LIN {X 0,Y 361.861,Z 153.411,A -85,B 0,C 180,E1 -12922.982,E2 -12922.982} C_VEL
LIN {X 0,Y 361.857,Z 153.413,A -85,B 0,C 180,E1 -12926.632,E2 -12926.632} C_VEL
LIN {X 0,Y 361.847,Z 153.408,A -85,B 0,C 180,E1 -12929.67,E2 -12929.67} C_VEL
LIN {X 0,Y 361.854,Z 153.407,A -85,B 0,C 180,E1 -12933.468,E2 -12933.468} C_VEL
LIN {X 0,Y 361.862,Z 153.407,A -85,B 0,C 180,E1 -12937.144,E2 -12937.144} C_VEL
LIN {X 0,Y 361.842,Z 153.411,A -85,B 0,C 180,E1 -12940.72,E2 -12940.72} C_VEL
LIN {X 0,Y 361.871,Z 153.406,A -85,B 0,C 180,E1 -12943.064,E2 -12943.064} C_VEL
LIN {X 0,Y 361.967,Z 153.396,A -85,B 0,C 180,E1 -12946.527,E2 -12946.527} C_VEL
LIN {X 0,Y 361.997,Z 153.394,A -85,B 0,C 180,E1 -12949.938,E2 -12949.938} C_VEL
LIN {X 0,Y 362.125,Z 153.374,A -85,B 0,C 180,E1 -12953.314,E2 -12953.314} C_VEL
LIN {X 0,Y 362.262,Z 153.362,A -85,B 0,C 180,E1 -12957.777,E2 -12957.777} C_VEL
LIN {X 0,Y 362.178,Z 153.368,A -85,B 0,C 180,E1 -12961.112,E2 -12961.112} C_VEL
LIN {X 0,Y 362.268,Z 153.358,A -85,B 0,C 180,E1 -12962.224,E2 -12962.224} C_VEL
LIN {X 0,Y 362.122,Z 153.374,A -85,B 0,C 180,E1 -12966.688,E2 -12966.688} C_VEL
LIN {X 0,Y 362.003,Z 153.391,A -85,B 0,C 180,E1 -12970.063,E2 -12970.063} C_VEL
LIN {X 0,Y 361.985,Z 153.394,A -85,B 0,C 180,E1 -12973.887,E2 -12973.887} C_VEL
LIN {X 0,Y 361.891,Z 153.403,A -85,B 0,C 180,E1 -12978.103,E2 -12978.103} C_VEL
LIN {X 0,Y 361.858,Z 153.41,A -85,B 0,C 180,E1 -12981.656,E2 -12981.656} C_VEL
LIN {X 0,Y 361.884,Z 153.409,A -85,B 0,C 180,E1 -12985.294,E2 -12985.294} C_VEL
LIN {X 0,Y 361.86,Z 153.413,A -85,B 0,C 180,E1 -12989.074,E2 -12989.074} C_VEL
LIN {X 0,Y 361.851,Z 153.414,A -85,B 0,C 180,E1 -12992.945,E2 -12992.945} C_VEL
LIN {X 0,Y 361.868,Z 153.406,A -85,B 0,C 180,E1 -12995.637,E2 -12995.637} C_VEL
LIN {X 0,Y 361.831,Z 153.415,A -85,B 0,C 180,E1 -12999.018,E2 -12999.018} C_VEL
LIN {X 0,Y 361.836,Z 153.415,A -85,B 0,C 180,E1 -13002.83,E2 -13002.83} C_VEL
LIN {X 0,Y 361.817,Z 153.412,A -85,B 0,C 180,E1 -13005.947,E2 -13005.947} C_VEL
LIN {X 0,Y 361.815,Z 153.413,A -85,B 0,C 180,E1 -13009.249,E2 -13009.249} C_VEL
LIN {X 0,Y 361.868,Z 153.408,A -85,B 0,C 180,E1 -13012.982,E2 -13012.982} C_VEL
LIN {X 0,Y 361.862,Z 153.411,A -85,B 0,C 180,E1 -13016.631,E2 -13016.631} C_VEL
LIN {X 0,Y 361.902,Z 153.409,A -85,B 0,C 180,E1 -13020.668,E2 -13020.668} C_VEL
LIN {X 0,Y 361.894,Z 153.433,A -85,B 0,C 180,E1 -13020.775,E2 -13020.775} C_VEL
LIN {X 0,Y 364.474,Z 166.518,A -85,B 0,C 180,E1 -13023.977,E2 -13023.977} C_VEL
LIN {X 0,Y 365.226,Z 170.606,A -85,B 0,C 180,E1 -13024.954,E2 -13024.954} C_VEL
LIN {X 0,Y 364.174,Z 182.944,A -85,B 0,C 180,E1 -13027.691,E2 -13027.691} C_VEL
LIN {X 0,Y 363.842,Z 187.528,A -85,B 0,C 180,E1 -13028.704,E2 -13028.704} C_VEL
LIN {X 0,Y 368.638,Z 221.989,A -85,B 0,C 180,E1 -13029.653,E2 -13029.653} C_VEL
LIN {X 0,Y 367.445,Z 296.055,A -85,B 0,C 180,E1 -13031.133,E2 -13031.133} C_VEL
LIN {X 0,Y 366.835,Z 309.281,A -85,B 0,C 180,E1 -13031.608,E2 -13031.608} C_VEL
LIN {X 0,Y 366.087,Z 321.461,A -85,B 0,C 180,E1 -13032.256,E2 -13032.256} C_VEL
LIN {X 0,Y 365.205,Z 332.949,A -85,B 0,C 180,E1 -13033.078,E2 -13033.078} C_VEL
LIN {X 0,Y 364.195,Z 344.752,A -85,B 0,C 180,E1 -13034.182,E2 -13034.182} C_VEL
LIN {X 0,Y 363.374,Z 355.364,A -85,B 0,C 180,E1 -13035.437,E2 -13035.437} C_VEL
LIN {X 0,Y 362.449,Z 364.896,A -85,B 0,C 180,E1 -13036.83,E2 -13036.83} C_VEL
LIN {X 0,Y 361.592,Z 374.066,A -85,B 0,C 180,E1 -13038.508,E2 -13038.508} C_VEL
LIN {X 0,Y 361.034,Z 381.452,A -85,B 0,C 180,E1 -13040.193,E2 -13040.193} C_VEL
LIN {X 0,Y 360.707,Z 386.445,A -85,B 0,C 180,E1 -13041.597,E2 -13041.597} C_VEL
LIN {X 0,Y 360.486,Z 391.284,A -85,B 0,C 180,E1 -13043.282,E2 -13043.282} C_VEL
LIN {X 0,Y 360.37,Z 394.981,A -85,B 0,C 180,E1 -13044.965,E2 -13044.965} C_VEL
LIN {X 0,Y 360.314,Z 397.642,A -85,B 0,C 180,E1 -13046.645,E2 -13046.645} C_VEL
LIN {X 0,Y 360.321,Z 398.891,A -85,B 0,C 180,E1 -13047.764,E2 -13047.764} C_VEL
LIN {X 0,Y 360.39,Z 399.729,A -85,B 0,C 180,E1 -13048.882,E2 -13048.882} C_VEL
LIN {X 0,Y 360.426,Z 400.127,A -85,B 0,C 180,E1 -13050,E2 -13050} C_VEL
LIN {X 0,Y 360.36,Z 400.131,A -85,B 0,C 180,E1 -13051.117,E2 -13051.117} C_VEL
LIN {X 0,Y 360.299,Z 398.972,A -85,B 0,C 180,E1 -13053.355,E2 -13053.355} C_VEL
LIN {X 0,Y 360.344,Z 397.756,A -85,B 0,C 180,E1 -13054.474,E2 -13054.474} C_VEL
LIN {X 0,Y 360.379,Z 395.538,A -85,B 0,C 180,E1 -13055.961,E2 -13055.961} C_VEL
LIN {X 0,Y 360.659,Z 391.599,A -85,B 0,C 180,E1 -13057.84,E2 -13057.84} C_VEL
LIN {X 0,Y 361.085,Z 386.927,A -85,B 0,C 180,E1 -13059.523,E2 -13059.523} C_VEL
LIN {X 0,Y 361.83,Z 379.903,A -85,B 0,C 180,E1 -13061.484,E2 -13061.484} C_VEL
LIN {X 0,Y 362.895,Z 372.328,A -85,B 0,C 180,E1 -13063.153,E2 -13063.153} C_VEL
LIN {X 0,Y 364.019,Z 363.164,A -85,B 0,C 180,E1 -13064.774,E2 -13064.774} C_VEL
LIN {X 0,Y 365.223,Z 353.139,A -85,B 0,C 180,E1 -13066.202,E2 -13066.202} C_VEL
LIN {X 0,Y 366.549,Z 342.34,A -85,B 0,C 180,E1 -13067.433,E2 -13067.433} C_VEL
LIN {X 0,Y 367.948,Z 330.06,A -85,B 0,C 180,E1 -13068.515,E2 -13068.515} C_VEL
LIN {X 0,Y 369.043,Z 318.085,A -85,B 0,C 180,E1 -13069.323,E2 -13069.323} C_VEL
LIN {X 0,Y 370.045,Z 304.955,A -85,B 0,C 180,E1 -13069.954,E2 -13069.954} C_VEL
LIN {X 0,Y 370.743,Z 291.887,A -85,B 0,C 180,E1 -13070.349,E2 -13070.349} C_VEL
LIN {X 0,Y 371.93,Z 221.499,A -85,B 0,C 180,E1 -13071.775,E2 -13071.775} C_VEL
LIN {X 0,Y 368.049,Z 198.796,A -85,B 0,C 180,E1 -13072.556,E2 -13072.556} C_VEL
LIN {X 0,Y 365.479,Z 186.6,A -85,B 0,C 180,E1 -13073.056,E2 -13073.056} C_VEL
LIN {X 0,Y 366.598,Z 175.915,A -85,B 0,C 180,E1 -13075.493,E2 -13075.493} C_VEL
LIN {X 0,Y 365.089,Z 167.35,A -85,B 0,C 180,E1 -13077.685,E2 -13077.685} C_VEL
LIN {X 0,Y 362.679,Z 156.746,A -85,B 0,C 180,E1 -13080.558,E2 -13080.558} C_VEL
LIN {X 0,Y 361.891,Z 153.408,A -85,B 0,C 180,E1 -13081.516,E2 -13081.516} C_VEL
LIN {X 0,Y 361.876,Z 153.407,A -85,B 0,C 180,E1 -13085.344,E2 -13085.344} C_VEL
LIN {X 0,Y 361.828,Z 153.418,A -85,B 0,C 180,E1 -13089.018,E2 -13089.018} C_VEL
LIN {X 0,Y 361.833,Z 153.416,A -85,B 0,C 180,E1 -13092.829,E2 -13092.829} C_VEL
LIN {X 0,Y 361.815,Z 153.414,A -85,B 0,C 180,E1 -13095.947,E2 -13095.947} C_VEL
LIN {X 0,Y 361.812,Z 153.414,A -85,B 0,C 180,E1 -13099.249,E2 -13099.249} C_VEL
LIN {X 0,Y 361.862,Z 153.409,A -85,B 0,C 180,E1 -13102.981,E2 -13102.981} C_VEL
LIN {X 0,Y 361.859,Z 153.408,A -85,B 0,C 180,E1 -13106.631,E2 -13106.631} C_VEL
LIN {X 0,Y 361.849,Z 153.404,A -85,B 0,C 180,E1 -13109.669,E2 -13109.669} C_VEL
LIN {X 0,Y 361.855,Z 153.401,A -85,B 0,C 180,E1 -13113.467,E2 -13113.467} C_VEL
LIN {X 0,Y 361.856,Z 153.399,A -85,B 0,C 180,E1 -13117.142,E2 -13117.142} C_VEL
LIN {X 0,Y 361.843,Z 153.408,A -85,B 0,C 180,E1 -13120.719,E2 -13120.719} C_VEL
LIN {X 0,Y 361.879,Z 153.403,A -85,B 0,C 180,E1 -13123.063,E2 -13123.063} C_VEL
LIN {X 0,Y 362.001,Z 153.382,A -85,B 0,C 180,E1 -13126.527,E2 -13126.527} C_VEL
LIN {X 0,Y 361.998,Z 153.393,A -85,B 0,C 180,E1 -13129.936,E2 -13129.936} C_VEL
LIN {X 0,Y 362.125,Z 153.371,A -85,B 0,C 180,E1 -13133.312,E2 -13133.312} C_VEL
LIN {X 0,Y 362.267,Z 153.353,A -85,B 0,C 180,E1 -13137.776,E2 -13137.776} C_VEL
LIN {X 0,Y 362.178,Z 153.362,A -85,B 0,C 180,E1 -13141.111,E2 -13141.111} C_VEL
LIN {X 0,Y 362.279,Z 153.353,A -85,B 0,C 180,E1 -13142.223,E2 -13142.223} C_VEL
LIN {X 0,Y 362.126,Z 153.369,A -85,B 0,C 180,E1 -13146.686,E2 -13146.686} C_VEL
LIN {X 0,Y 362.002,Z 153.383,A -85,B 0,C 180,E1 -13150.062,E2 -13150.062} C_VEL
LIN {X 0,Y 361.999,Z 153.386,A -85,B 0,C 180,E1 -13153.898,E2 -13153.898} C_VEL
LIN {X 0,Y 361.929,Z 153.404,A -85,B 0,C 180,E1 -13156.933,E2 -13156.933} C_VEL
LIN {X 0,Y 361.887,Z 153.408,A -85,B 0,C 180,E1 -13160.46,E2 -13160.46} C_VEL
LIN {X 0,Y 361.893,Z 153.407,A -85,B 0,C 180,E1 -13164.112,E2 -13164.112} C_VEL
LIN {X 0,Y 361.941,Z 153.405,A -85,B 0,C 180,E1 -13166.721,E2 -13166.721} C_VEL
LIN {X 0,Y 361.874,Z 153.408,A -85,B 0,C 180,E1 -13170.327,E2 -13170.327} C_VEL
LIN {X 0,Y 361.853,Z 153.413,A -85,B 0,C 180,E1 -13174.28,E2 -13174.28} C_VEL
LIN {X 0,Y 361.862,Z 153.414,A -85,B 0,C 180,E1 -13177.222,E2 -13177.222} C_VEL
LIN {X 0,Y 361.834,Z 153.421,A -85,B 0,C 180,E1 -13180.755,E2 -13180.755} C_VEL
LIN {X 0,Y 361.877,Z 153.565,A -85,B 0,C 180,E1 -13183.963,E2 -13183.963} C_VEL
LIN {X 0,Y 364.155,Z 163.607,A -85,B 0,C 180,E1 -13186.916,E2 -13186.916} C_VEL
LIN {X 0,Y 369.825,Z 177.061,A -85,B 0,C 180,E1 -13187.659,E2 -13187.659} C_VEL
LIN {X 0,Y 372.692,Z 189.395,A -85,B 0,C 180,E1 -13188.144,E2 -13188.144} C_VEL
LIN {X 0,Y 370.937,Z 271.319,A -85,B 0,C 180,E1 -13189.805,E2 -13189.805} C_VEL
LIN {X 0,Y 370.285,Z 284.163,A -85,B 0,C 180,E1 -13190.276,E2 -13190.276} C_VEL
LIN {X 0,Y 369.554,Z 296.511,A -85,B 0,C 180,E1 -13190.953,E2 -13190.953} C_VEL
LIN {X 0,Y 368.588,Z 307.524,A -85,B 0,C 180,E1 -13191.754,E2 -13191.754} C_VEL
LIN {X 0,Y 367.447,Z 318.475,A -85,B 0,C 180,E1 -13192.78,E2 -13192.78} C_VEL
LIN {X 0,Y 366.247,Z 329.044,A -85,B 0,C 180,E1 -13194.027,E2 -13194.027} C_VEL
LIN {X 0,Y 365.011,Z 338.404,A -85,B 0,C 180,E1 -13195.389,E2 -13195.389} C_VEL
LIN {X 0,Y 363.9,Z 346.954,A -85,B 0,C 180,E1 -13196.935,E2 -13196.935} C_VEL
LIN {X 0,Y 362.763,Z 355.098,A -85,B 0,C 180,E1 -13198.786,E2 -13198.786} C_VEL
LIN {X 0,Y 362.019,Z 360.516,A -85,B 0,C 180,E1 -13200.328,E2 -13200.328} C_VEL
LIN {X 0,Y 361.328,Z 365.639,A -85,B 0,C 180,E1 -13202.172,E2 -13202.172} C_VEL
LIN {X 0,Y 360.95,Z 368.647,A -85,B 0,C 180,E1 -13203.591,E2 -13203.591} C_VEL
LIN {X 0,Y 360.697,Z 370.391,A -85,B 0,C 180,E1 -13204.618,E2 -13204.618} C_VEL
LIN {X 0,Y 360.442,Z 372.569,A -85,B 0,C 180,E1 -13206.406,E2 -13206.406} C_VEL
LIN {X 0,Y 360.236,Z 373.739,A -85,B 0,C 180,E1 -13208.243,E2 -13208.243} C_VEL
LIN {X 0,Y 360.228,Z 373.938,A -85,B 0,C 180,E1 -13209.465,E2 -13209.465} C_VEL
LIN {X 0,Y 360.193,Z 373.659,A -85,B 0,C 180,E1 -13210.628,E2 -13210.628} C_VEL
LIN {X 0,Y 360.293,Z 371.928,A -85,B 0,C 180,E1 -13212.901,E2 -13212.901} C_VEL
LIN {X 0,Y 360.531,Z 369.267,A -85,B 0,C 180,E1 -13214.742,E2 -13214.742} C_VEL
LIN {X 0,Y 360.897,Z 364.776,A -85,B 0,C 180,E1 -13216.823,E2 -13216.823} C_VEL
LIN {X 0,Y 361.319,Z 359.013,A -85,B 0,C 180,E1 -13218.784,E2 -13218.784} C_VEL
LIN {X 0,Y 361.905,Z 352.492,A -85,B 0,C 180,E1 -13220.499,E2 -13220.499} C_VEL
LIN {X 0,Y 362.633,Z 344.333,A -85,B 0,C 180,E1 -13222.203,E2 -13222.203} C_VEL
LIN {X 0,Y 363.424,Z 335.995,A -85,B 0,C 180,E1 -13223.616,E2 -13223.616} C_VEL
LIN {X 0,Y 364.387,Z 325.786,A -85,B 0,C 180,E1 -13225.021,E2 -13225.021} C_VEL
LIN {X 0,Y 365.377,Z 314.188,A -85,B 0,C 180,E1 -13226.278,E2 -13226.278} C_VEL
LIN {X 0,Y 366.165,Z 302.906,A -85,B 0,C 180,E1 -13227.244,E2 -13227.244} C_VEL
LIN {X 0,Y 366.78,Z 291.305,A -85,B 0,C 180,E1 -13228.01,E2 -13228.01} C_VEL
LIN {X 0,Y 367.353,Z 278.024,A -85,B 0,C 180,E1 -13228.63,E2 -13228.63} C_VEL
LIN {X 0,Y 367.735,Z 264.328,A -85,B 0,C 180,E1 -13229.027,E2 -13229.027} C_VEL
LIN {X 0,Y 368.978,Z 187.085,A -85,B 0,C 180,E1 -13230.546,E2 -13230.546} C_VEL
LIN {X 0,Y 365.057,Z 166.996,A -85,B 0,C 180,E1 -13231.152,E2 -13231.152} C_VEL
LIN {X 0,Y 363.773,Z 162.901,A -85,B 0,C 180,E1 -13231.315,E2 -13231.315} C_VEL
LIN {X 0,Y 362.669,Z 156.347,A -85,B 0,C 180,E1 -13233.055,E2 -13233.055} C_VEL
LIN {X 0,Y 361.939,Z 153.406,A -85,B 0,C 180,E1 -13233.897,E2 -13233.897} C_VEL
LIN {X 0,Y 361.945,Z 153.396,A -85,B 0,C 180,E1 -13234.765,E2 -13234.765} C_VEL
LIN {X 0,Y 361.37,Z 153.472,A -85,B 0,C 180,E1 -13235.695,E2 -13235.695} C_VEL
LIN {X 0,Y 358.557,Z 153.819,A -85,B 0,C 180,E1 -13237.209,E2 -13237.209} C_VEL
LIN {X 0,Y 356.11,Z 154.124,A -85,B 0,C 180,E1 -13238.433,E2 -13238.433} C_VEL
LIN {X 0,Y 355.041,Z 154.258,A -85,B 0,C 180,E1 -13239.38,E2 -13239.38} C_VEL
LIN {X 0,Y 354.948,Z 154.267,A -85,B 0,C 180,E1 -13239.701,E2 -13239.701} C_VEL
LIN {X 0,Y 354.893,Z 154.275,A -85,B 0,C 180,E1 -13242.582,E2 -13242.582} C_VEL
LIN {X 0,Y 354.823,Z 154.285,A -85,B 0,C 180,E1 -13246.099,E2 -13246.099} C_VEL
LIN {X 0,Y 354.816,Z 154.284,A -85,B 0,C 180,E1 -13248.477,E2 -13248.477} C_VEL
LIN {X 0,Y 354.795,Z 154.288,A -85,B 0,C 180,E1 -13252.109,E2 -13252.109} C_VEL
LIN {X 0,Y 354.79,Z 154.29,A -85,B 0,C 180,E1 -13255.836,E2 -13255.836} C_VEL
LIN {X 0,Y 354.79,Z 154.29,A -85,B 0,C 180,E1 -13259.685,E2 -13259.685} C_VEL
LIN {X 0,Y 354.783,Z 154.288,A -85,B 0,C 180,E1 -13262.334,E2 -13262.334} C_VEL
LIN {X 0,Y 354.815,Z 154.286,A -85,B 0,C 180,E1 -13265.699,E2 -13265.699} C_VEL
LIN {X 0,Y 354.766,Z 154.293,A -85,B 0,C 180,E1 -13269.413,E2 -13269.413} C_VEL
LIN {X 0,Y 354.779,Z 154.293,A -85,B 0,C 180,E1 -13272.867,E2 -13272.867} C_VEL
LIN {X 0,Y 354.761,Z 154.291,A -85,B 0,C 180,E1 -13276.104,E2 -13276.104} C_VEL
LIN {X 0,Y 354.762,Z 154.294,A -85,B 0,C 180,E1 -13279.176,E2 -13279.176} C_VEL
LIN {X 0,Y 354.798,Z 154.289,A -85,B 0,C 180,E1 -13282.405,E2 -13282.405} C_VEL
LIN {X 0,Y 354.807,Z 154.289,A -85,B 0,C 180,E1 -13284.941,E2 -13284.941} C_VEL
LIN {X 0,Y 354.793,Z 154.291,A -85,B 0,C 180,E1 -13288.406,E2 -13288.406} C_VEL
LIN {X 0,Y 354.789,Z 154.288,A -85,B 0,C 180,E1 -13291.614,E2 -13291.614} C_VEL
LIN {X 0,Y 354.803,Z 154.286,A -85,B 0,C 180,E1 -13295.42,E2 -13295.42} C_VEL
LIN {X 0,Y 354.819,Z 154.284,A -85,B 0,C 180,E1 -13299.113,E2 -13299.113} C_VEL
LIN {X 0,Y 354.839,Z 154.283,A -85,B 0,C 180,E1 -13302.718,E2 -13302.718} C_VEL
LIN {X 0,Y 354.911,Z 154.278,A -85,B 0,C 180,E1 -13306.254,E2 -13306.254} C_VEL
LIN {X 0,Y 354.953,Z 154.27,A -85,B 0,C 180,E1 -13309.736,E2 -13309.736} C_VEL
LIN {X 0,Y 355.092,Z 154.25,A -85,B 0,C 180,E1 -13313.181,E2 -13313.181} C_VEL
LIN {X 0,Y 355.223,Z 154.238,A -85,B 0,C 180,E1 -13317.733,E2 -13317.733} C_VEL
LIN {X 0,Y 355.149,Z 154.243,A -85,B 0,C 180,E1 -13321.135,E2 -13321.135} C_VEL
LIN {X 0,Y 355.23,Z 154.234,A -85,B 0,C 180,E1 -13322.268,E2 -13322.268} C_VEL
LIN {X 0,Y 355.088,Z 154.25,A -85,B 0,C 180,E1 -13326.821,E2 -13326.821} C_VEL
LIN {X 0,Y 354.959,Z 154.267,A -85,B 0,C 180,E1 -13330.265,E2 -13330.265} C_VEL
LIN {X 0,Y 354.928,Z 154.272,A -85,B 0,C 180,E1 -13334.006,E2 -13334.006} C_VEL
LIN {X 0,Y 354.849,Z 154.281,A -85,B 0,C 180,E1 -13338.07,E2 -13338.07} C_VEL
LIN {X 0,Y 354.811,Z 154.285,A -85,B 0,C 180,E1 -13342.108,E2 -13342.108} C_VEL
LIN {X 0,Y 354.853,Z 154.28,A -85,B 0,C 180,E1 -13344.577,E2 -13344.577} C_VEL
LIN {X 0,Y 354.801,Z 154.286,A -85,B 0,C 180,E1 -13348.386,E2 -13348.386} C_VEL
LIN {X 0,Y 354.789,Z 154.288,A -85,B 0,C 180,E1 -13352.334,E2 -13352.334} C_VEL
LIN {X 0,Y 354.823,Z 154.284,A -85,B 0,C 180,E1 -13355.698,E2 -13355.698} C_VEL
LIN {X 0,Y 354.772,Z 154.291,A -85,B 0,C 180,E1 -13359.413,E2 -13359.413} C_VEL
LIN {X 0,Y 354.788,Z 154.293,A -85,B 0,C 180,E1 -13362.866,E2 -13362.866} C_VEL
LIN {X 0,Y 354.767,Z 154.291,A -85,B 0,C 180,E1 -13366.103,E2 -13366.103} C_VEL
LIN {X 0,Y 354.768,Z 154.291,A -85,B 0,C 180,E1 -13369.176,E2 -13369.176} C_VEL
LIN {X 0,Y 354.804,Z 154.291,A -85,B 0,C 180,E1 -13372.404,E2 -13372.404} C_VEL
LIN {X 0,Y 354.815,Z 154.286,A -85,B 0,C 180,E1 -13374.941,E2 -13374.941} C_VEL
LIN {X 0,Y 354.797,Z 154.293,A -85,B 0,C 180,E1 -13378.405,E2 -13378.405} C_VEL
LIN {X 0,Y 354.876,Z 154.373,A -85,B 0,C 180,E1 -13380.53,E2 -13380.53} C_VEL
LIN {X 0,Y 357.397,Z 167.225,A -85,B 0,C 180,E1 -13383.739,E2 -13383.739} C_VEL
LIN {X 0,Y 358.221,Z 172.67,A -85,B 0,C 180,E1 -13385.051,E2 -13385.051} C_VEL
LIN {X 0,Y 356.892,Z 187.314,A -85,B 0,C 180,E1 -13388.356,E2 -13388.356} C_VEL
LIN {X 0,Y 361.844,Z 223.24,A -85,B 0,C 180,E1 -13389.355,E2 -13389.355} C_VEL
LIN {X 0,Y 360.61,Z 295.988,A -85,B 0,C 180,E1 -13390.836,E2 -13390.836} C_VEL
LIN {X 0,Y 359.993,Z 309.152,A -85,B 0,C 180,E1 -13391.319,E2 -13391.319} C_VEL
LIN {X 0,Y 359.213,Z 321.297,A -85,B 0,C 180,E1 -13391.978,E2 -13391.978} C_VEL
LIN {X 0,Y 358.23,Z 333.568,A -85,B 0,C 180,E1 -13392.885,E2 -13392.885} C_VEL
LIN {X 0,Y 357.186,Z 345.199,A -85,B 0,C 180,E1 -13394.01,E2 -13394.01} C_VEL
LIN {X 0,Y 356.369,Z 355.446,A -85,B 0,C 180,E1 -13395.258,E2 -13395.258} C_VEL
LIN {X 0,Y 355.482,Z 364.242,A -85,B 0,C 180,E1 -13396.567,E2 -13396.567} C_VEL
LIN {X 0,Y 354.764,Z 372.124,A -85,B 0,C 180,E1 -13397.994,E2 -13397.994} C_VEL
LIN {X 0,Y 354.106,Z 379.808,A -85,B 0,C 180,E1 -13399.71,E2 -13399.71} C_VEL
LIN {X 0,Y 353.651,Z 385.979,A -85,B 0,C 180,E1 -13401.428,E2 -13401.428} C_VEL
LIN {X 0,Y 353.397,Z 390.862,A -85,B 0,C 180,E1 -13403.147,E2 -13403.147} C_VEL
LIN {X 0,Y 353.273,Z 394.6,A -85,B 0,C 180,E1 -13404.864,E2 -13404.864} C_VEL
LIN {X 0,Y 353.237,Z 397.301,A -85,B 0,C 180,E1 -13406.578,E2 -13406.578} C_VEL
LIN {X 0,Y 353.225,Z 398.568,A -85,B 0,C 180,E1 -13407.719,E2 -13407.719} C_VEL
LIN {X 0,Y 353.292,Z 399.434,A -85,B 0,C 180,E1 -13408.86,E2 -13408.86} C_VEL
LIN {X 0,Y 353.33,Z 399.858,A -85,B 0,C 180,E1 -13410,E2 -13410} C_VEL
LIN {X 0,Y 353.261,Z 399.878,A -85,B 0,C 180,E1 -13411.14,E2 -13411.14} C_VEL
LIN {X 0,Y 353.22,Z 398.762,A -85,B 0,C 180,E1 -13413.422,E2 -13413.422} C_VEL
LIN {X 0,Y 353.257,Z 397.574,A -85,B 0,C 180,E1 -13414.564,E2 -13414.564} C_VEL
LIN {X 0,Y 353.274,Z 395.664,A -85,B 0,C 180,E1 -13415.899,E2 -13415.899} C_VEL
LIN {X 0,Y 353.608,Z 391.49,A -85,B 0,C 180,E1 -13417.997,E2 -13417.997} C_VEL
LIN {X 0,Y 354.05,Z 386.871,A -85,B 0,C 180,E1 -13419.714,E2 -13419.714} C_VEL
LIN {X 0,Y 354.861,Z 379.914,A -85,B 0,C 180,E1 -13421.712,E2 -13421.712} C_VEL
LIN {X 0,Y 355.97,Z 372.413,A -85,B 0,C 180,E1 -13423.414,E2 -13423.414} C_VEL
LIN {X 0,Y 357.098,Z 363.665,A -85,B 0,C 180,E1 -13425.019,E2 -13425.019} C_VEL
LIN {X 0,Y 358.412,Z 353.438,A -85,B 0,C 180,E1 -13426.518,E2 -13426.518} C_VEL
LIN {X 0,Y 359.796,Z 342.763,A -85,B 0,C 180,E1 -13427.771,E2 -13427.771} C_VEL
LIN {X 0,Y 361.062,Z 332.443,A -85,B 0,C 180,E1 -13428.734,E2 -13428.734} C_VEL
LIN {X 0,Y 362.288,Z 320.121,A -85,B 0,C 180,E1 -13429.624,E2 -13429.624} C_VEL
LIN {X 0,Y 363.392,Z 307.201,A -85,B 0,C 180,E1 -13430.298,E2 -13430.298} C_VEL
LIN {X 0,Y 364.193,Z 294.662,A -85,B 0,C 180,E1 -13430.731,E2 -13430.731} C_VEL
LIN {X 0,Y 365.577,Z 222.876,A -85,B 0,C 180,E1 -13432.217,E2 -13432.217} C_VEL
LIN {X 0,Y 361.997,Z 201.712,A -85,B 0,C 180,E1 -13432.961,E2 -13432.961} C_VEL
LIN {X 0,Y 358.807,Z 186.375,A -85,B 0,C 180,E1 -13433.584,E2 -13433.584} C_VEL
LIN {X 0,Y 359.748,Z 177.066,A -85,B 0,C 180,E1 -13435.762,E2 -13435.762} C_VEL
LIN {X 0,Y 358.053,Z 168.195,A -85,B 0,C 180,E1 -13438.104,E2 -13438.104} C_VEL
LIN {X 0,Y 355.749,Z 158.105,A -85,B 0,C 180,E1 -13440.907,E2 -13440.907} C_VEL
LIN {X 0,Y 354.852,Z 154.282,A -85,B 0,C 180,E1 -13442.018,E2 -13442.018} C_VEL
LIN {X 0,Y 354.823,Z 154.289,A -85,B 0,C 180,E1 -13445.699,E2 -13445.699} C_VEL
LIN {X 0,Y 354.77,Z 154.294,A -85,B 0,C 180,E1 -13449.412,E2 -13449.412} C_VEL
LIN {X 0,Y 354.785,Z 154.294,A -85,B 0,C 180,E1 -13452.866,E2 -13452.866} C_VEL
LIN {X 0,Y 354.765,Z 154.293,A -85,B 0,C 180,E1 -13456.103,E2 -13456.103} C_VEL
LIN {X 0,Y 354.765,Z 154.291,A -85,B 0,C 180,E1 -13459.175,E2 -13459.175} C_VEL
LIN {X 0,Y 354.8,Z 154.285,A -85,B 0,C 180,E1 -13462.404,E2 -13462.404} C_VEL
LIN {X 0,Y 354.809,Z 154.284,A -85,B 0,C 180,E1 -13464.94,E2 -13464.94} C_VEL
LIN {X 0,Y 354.795,Z 154.287,A -85,B 0,C 180,E1 -13468.405,E2 -13468.405} C_VEL
LIN {X 0,Y 354.798,Z 154.287,A -85,B 0,C 180,E1 -13471.614,E2 -13471.614} C_VEL
LIN {X 0,Y 354.806,Z 154.286,A -85,B 0,C 180,E1 -13475.419,E2 -13475.419} C_VEL
LIN {X 0,Y 354.817,Z 154.285,A -85,B 0,C 180,E1 -13479.112,E2 -13479.112} C_VEL
LIN {X 0,Y 354.846,Z 154.278,A -85,B 0,C 180,E1 -13482.717,E2 -13482.717} C_VEL
LIN {X 0,Y 354.942,Z 154.263,A -85,B 0,C 180,E1 -13486.254,E2 -13486.254} C_VEL
LIN {X 0,Y 354.955,Z 154.271,A -85,B 0,C 180,E1 -13489.735,E2 -13489.735} C_VEL
LIN {X 0,Y 355.09,Z 154.247,A -85,B 0,C 180,E1 -13493.179,E2 -13493.179} C_VEL
LIN {X 0,Y 355.229,Z 154.229,A -85,B 0,C 180,E1 -13497.732,E2 -13497.732} C_VEL
LIN {X 0,Y 355.149,Z 154.237,A -85,B 0,C 180,E1 -13501.133,E2 -13501.133} C_VEL
LIN {X 0,Y 355.242,Z 154.23,A -85,B 0,C 180,E1 -13502.267,E2 -13502.267} C_VEL
LIN {X 0,Y 355.091,Z 154.246,A -85,B 0,C 180,E1 -13506.819,E2 -13506.819} C_VEL
LIN {X 0,Y 354.958,Z 154.26,A -85,B 0,C 180,E1 -13510.264,E2 -13510.264} C_VEL
LIN {X 0,Y 354.944,Z 154.265,A -85,B 0,C 180,E1 -13514.018,E2 -13514.018} C_VEL
LIN {X 0,Y 354.89,Z 154.272,A -85,B 0,C 180,E1 -13518.091,E2 -13518.091} C_VEL
LIN {X 0,Y 354.819,Z 154.282,A -85,B 0,C 180,E1 -13521.417,E2 -13521.417} C_VEL
LIN {X 0,Y 354.86,Z 154.282,A -85,B 0,C 180,E1 -13524.576,E2 -13524.576} C_VEL
LIN {X 0,Y 354.882,Z 154.28,A -85,B 0,C 180,E1 -13527.095,E2 -13527.095} C_VEL
LIN {X 0,Y 354.853,Z 154.283,A -85,B 0,C 180,E1 -13529.678,E2 -13529.678} C_VEL
LIN {X 0,Y 354.805,Z 154.289,A -85,B 0,C 180,E1 -13533.701,E2 -13533.701} C_VEL
LIN {X 0,Y 354.796,Z 154.293,A -85,B 0,C 180,E1 -13536.459,E2 -13536.459} C_VEL
LIN {X 0,Y 354.822,Z 154.286,A -85,B 0,C 180,E1 -13539.423,E2 -13539.423} C_VEL
LIN {X 0,Y 354.845,Z 154.439,A -85,B 0,C 180,E1 -13543.462,E2 -13543.462} C_VEL
LIN {X 0,Y 357.055,Z 163.923,A -85,B 0,C 180,E1 -13546.329,E2 -13546.329} C_VEL
LIN {X 0,Y 363.741,Z 179.666,A -85,B 0,C 180,E1 -13547.24,E2 -13547.24} C_VEL
LIN {X 0,Y 366.304,Z 190.505,A -85,B 0,C 180,E1 -13547.681,E2 -13547.681} C_VEL
LIN {X 0,Y 364.472,Z 271.592,A -85,B 0,C 180,E1 -13549.353,E2 -13549.353} C_VEL
LIN {X 0,Y 363.85,Z 284.02,A -85,B 0,C 180,E1 -13549.814,E2 -13549.814} C_VEL
LIN {X 0,Y 363.09,Z 296.227,A -85,B 0,C 180,E1 -13550.487,E2 -13550.487} C_VEL
LIN {X 0,Y 362.02,Z 307.908,A -85,B 0,C 180,E1 -13551.344,E2 -13551.344} C_VEL
LIN {X 0,Y 360.706,Z 319.796,A -85,B 0,C 180,E1 -13552.492,E2 -13552.492} C_VEL
LIN {X 0,Y 359.414,Z 330.433,A -85,B 0,C 180,E1 -13553.793,E2 -13553.793} C_VEL
LIN {X 0,Y 358.293,Z 338.41,A -85,B 0,C 180,E1 -13554.988,E2 -13554.988} C_VEL
LIN {X 0,Y 357.111,Z 347.022,A -85,B 0,C 180,E1 -13556.561,E2 -13556.561} C_VEL
LIN {X 0,Y 356.107,Z 353.716,A -85,B 0,C 180,E1 -13558.062,E2 -13558.062} C_VEL
LIN {X 0,Y 355.227,Z 359.657,A -85,B 0,C 180,E1 -13559.701,E2 -13559.701} C_VEL
LIN {X 0,Y 354.454,Z 365.017,A -85,B 0,C 180,E1 -13561.584,E2 -13561.584} C_VEL
LIN {X 0,Y 353.95,Z 368.768,A -85,B 0,C 180,E1 -13563.317,E2 -13563.317} C_VEL
LIN {X 0,Y 353.51,Z 371.835,A -85,B 0,C 180,E1 -13565.324,E2 -13565.324} C_VEL
LIN {X 0,Y 353.332,Z 373.104,A -85,B 0,C 180,E1 -13566.559,E2 -13566.559} C_VEL
LIN {X 0,Y 353.19,Z 373.857,A -85,B 0,C 180,E1 -13567.786,E2 -13567.786} C_VEL
LIN {X 0,Y 353.147,Z 374.205,A -85,B 0,C 180,E1 -13569.282,E2 -13569.282} C_VEL
LIN {X 0,Y 353.101,Z 373.47,A -85,B 0,C 180,E1 -13571.43,E2 -13571.43} C_VEL
LIN {X 0,Y 353.195,Z 372.315,A -85,B 0,C 180,E1 -13572.767,E2 -13572.767} C_VEL
LIN {X 0,Y 353.298,Z 371.008,A -85,B 0,C 180,E1 -13573.83,E2 -13573.83} C_VEL
LIN {X 0,Y 353.621,Z 367.944,A -85,B 0,C 180,E1 -13575.615,E2 -13575.615} C_VEL
LIN {X 0,Y 353.925,Z 363.798,A -85,B 0,C 180,E1 -13577.383,E2 -13577.383} C_VEL
LIN {X 0,Y 354.422,Z 357.408,A -85,B 0,C 180,E1 -13579.431,E2 -13579.431} C_VEL
LIN {X 0,Y 355.026,Z 350.686,A -85,B 0,C 180,E1 -13581.12,E2 -13581.12} C_VEL
LIN {X 0,Y 355.74,Z 343.324,A -85,B 0,C 180,E1 -13582.622,E2 -13582.622} C_VEL
LIN {X 0,Y 356.586,Z 334.719,A -85,B 0,C 180,E1 -13584.061,E2 -13584.061} C_VEL
LIN {X 0,Y 357.636,Z 324.029,A -85,B 0,C 180,E1 -13585.492,E2 -13585.492} C_VEL
LIN {X 0,Y 358.642,Z 312.376,A -85,B 0,C 180,E1 -13586.733,E2 -13586.733} C_VEL
LIN {X 0,Y 359.416,Z 300.812,A -85,B 0,C 180,E1 -13587.688,E2 -13587.688} C_VEL
LIN {X 0,Y 360.133,Z 288.368,A -85,B 0,C 180,E1 -13588.463,E2 -13588.463} C_VEL
LIN {X 0,Y 360.637,Z 275.636,A -85,B 0,C 180,E1 -13589.023,E2 -13589.023} C_VEL
LIN {X 0,Y 360.993,Z 260.577,A -85,B 0,C 180,E1 -13589.408,E2 -13589.408} C_VEL
LIN {X 0,Y 362.223,Z 188.056,A -85,B 0,C 180,E1 -13590.858,E2 -13590.858} C_VEL
LIN {X 0,Y 358.417,Z 168.827,A -85,B 0,C 180,E1 -13591.455,E2 -13591.455} C_VEL
LIN {X 0,Y 356.667,Z 163.075,A -85,B 0,C 180,E1 -13591.695,E2 -13591.695} C_VEL
LIN {X 0,Y 355.473,Z 156.829,A -85,B 0,C 180,E1 -13593.401,E2 -13593.401} C_VEL
LIN {X 0,Y 354.893,Z 154.279,A -85,B 0,C 180,E1 -13594.117,E2 -13594.117} C_VEL
LIN {X 0,Y 355.082,Z 154.251,A -85,B 0,C 180,E1 -13596.821,E2 -13596.821} C_VEL
LIN {X 0,Y 354.948,Z 154.267,A -85,B 0,C 180,E1 -13599.701,E2 -13599.701} C_VEL
LIN {X 0,Y 354.262,Z 154.355,A -85,B 0,C 180,E1 -13600.649,E2 -13600.649} C_VEL
LIN {X 0,Y 351.388,Z 154.713,A -85,B 0,C 180,E1 -13602.189,E2 -13602.189} C_VEL
LIN {X 0,Y 348.954,Z 155.017,A -85,B 0,C 180,E1 -13603.435,E2 -13603.435} C_VEL
LIN {X 0,Y 347.897,Z 155.147,A -85,B 0,C 180,E1 -13604.399,E2 -13604.399} C_VEL
LIN {X 0,Y 347.804,Z 155.158,A -85,B 0,C 180,E1 -13604.726,E2 -13604.726} C_VEL
LIN {X 0,Y 347.783,Z 155.161,A -85,B 0,C 180,E1 -13608.239,E2 -13608.239} C_VEL
LIN {X 0,Y 347.754,Z 155.169,A -85,B 0,C 180,E1 -13611.623,E2 -13611.623} C_VEL
LIN {X 0,Y 347.729,Z 155.17,A -85,B 0,C 180,E1 -13615.115,E2 -13615.115} C_VEL
LIN {X 0,Y 347.721,Z 155.171,A -85,B 0,C 180,E1 -13617.702,E2 -13617.702} C_VEL
LIN {X 0,Y 347.733,Z 155.167,A -85,B 0,C 180,E1 -13620.35,E2 -13620.35} C_VEL
LIN {X 0,Y 347.745,Z 155.165,A -85,B 0,C 180,E1 -13624.044,E2 -13624.044} C_VEL
LIN {X 0,Y 347.752,Z 155.169,A -85,B 0,C 180,E1 -13627.323,E2 -13627.323} C_VEL
LIN {X 0,Y 347.694,Z 155.172,A -85,B 0,C 180,E1 -13630.303,E2 -13630.303} C_VEL
LIN {X 0,Y 347.719,Z 155.17,A -85,B 0,C 180,E1 -13633.409,E2 -13633.409} C_VEL
LIN {X 0,Y 347.721,Z 155.172,A -85,B 0,C 180,E1 -13636.688,E2 -13636.688} C_VEL
LIN {X 0,Y 347.7,Z 155.171,A -85,B 0,C 180,E1 -13640.183,E2 -13640.183} C_VEL
LIN {X 0,Y 347.754,Z 155.169,A -85,B 0,C 180,E1 -13642.679,E2 -13642.679} C_VEL
LIN {X 0,Y 347.748,Z 155.165,A -85,B 0,C 180,E1 -13645.957,E2 -13645.957} C_VEL
LIN {X 0,Y 347.736,Z 155.166,A -85,B 0,C 180,E1 -13649.652,E2 -13649.652} C_VEL
LIN {X 0,Y 347.732,Z 155.167,A -85,B 0,C 180,E1 -13653.6,E2 -13653.6} C_VEL
LIN {X 0,Y 347.749,Z 155.168,A -85,B 0,C 180,E1 -13656.16,E2 -13656.16} C_VEL
LIN {X 0,Y 347.741,Z 155.168,A -85,B 0,C 180,E1 -13659.906,E2 -13659.906} C_VEL
LIN {X 0,Y 347.799,Z 155.164,A -85,B 0,C 180,E1 -13662.356,E2 -13662.356} C_VEL
LIN {X 0,Y 347.854,Z 155.155,A -85,B 0,C 180,E1 -13665.97,E2 -13665.97} C_VEL
LIN {X 0,Y 347.892,Z 155.148,A -85,B 0,C 180,E1 -13669.525,E2 -13669.525} C_VEL
LIN {X 0,Y 348.062,Z 155.126,A -85,B 0,C 180,E1 -13673.042,E2 -13673.042} C_VEL
LIN {X 0,Y 348.185,Z 155.114,A -85,B 0,C 180,E1 -13677.687,E2 -13677.687} C_VEL
LIN {X 0,Y 348.12,Z 155.119,A -85,B 0,C 180,E1 -13681.157,E2 -13681.157} C_VEL
LIN {X 0,Y 348.191,Z 155.111,A -85,B 0,C 180,E1 -13682.314,E2 -13682.314} C_VEL
LIN {X 0,Y 348.056,Z 155.127,A -85,B 0,C 180,E1 -13686.959,E2 -13686.959} C_VEL
LIN {X 0,Y 347.899,Z 155.146,A -85,B 0,C 180,E1 -13690.476,E2 -13690.476} C_VEL
LIN {X 0,Y 347.884,Z 155.148,A -85,B 0,C 180,E1 -13694.137,E2 -13694.137} C_VEL
LIN {X 0,Y 347.799,Z 155.158,A -85,B 0,C 180,E1 -13698.242,E2 -13698.242} C_VEL
LIN {X 0,Y 347.768,Z 155.165,A -85,B 0,C 180,E1 -13701.625,E2 -13701.625} C_VEL
LIN {X 0,Y 347.771,Z 155.167,A -85,B 0,C 180,E1 -13705.112,E2 -13705.112} C_VEL
LIN {X 0,Y 347.748,Z 155.17,A -85,B 0,C 180,E1 -13709.016,E2 -13709.016} C_VEL
LIN {X 0,Y 347.74,Z 155.166,A -85,B 0,C 180,E1 -13711.913,E2 -13711.913} C_VEL
LIN {X 0,Y 347.789,Z 155.16,A -85,B 0,C 180,E1 -13715.876,E2 -13715.876} C_VEL
LIN {X 0,Y 347.735,Z 155.172,A -85,B 0,C 180,E1 -13718.796,E2 -13718.796} C_VEL
LIN {X 0,Y 347.747,Z 155.165,A -85,B 0,C 180,E1 -13721.831,E2 -13721.831} C_VEL
LIN {X 0,Y 347.705,Z 155.173,A -85,B 0,C 180,E1 -13725.028,E2 -13725.028} C_VEL
LIN {X 0,Y 347.743,Z 155.169,A -85,B 0,C 180,E1 -13728.399,E2 -13728.399} C_VEL
LIN {X 0,Y 347.76,Z 155.168,A -85,B 0,C 180,E1 -13732.678,E2 -13732.678} C_VEL
LIN {X 0,Y 347.752,Z 155.166,A -85,B 0,C 180,E1 -13735.956,E2 -13735.956} C_VEL
LIN {X 0,Y 347.798,Z 155.164,A -85,B 0,C 180,E1 -13740.045,E2 -13740.045} C_VEL
LIN {X 0,Y 347.874,Z 155.453,A -85,B 0,C 180,E1 -13740.311,E2 -13740.311} C_VEL
LIN {X 0,Y 350.309,Z 167.904,A -85,B 0,C 180,E1 -13743.488,E2 -13743.488} C_VEL
LIN {X 0,Y 351.231,Z 172.968,A -85,B 0,C 180,E1 -13744.744,E2 -13744.744} C_VEL
LIN {X 0,Y 350.188,Z 184.489,A -85,B 0,C 180,E1 -13747.397,E2 -13747.397} C_VEL
LIN {X 0,Y 349.959,Z 186.998,A -85,B 0,C 180,E1 -13747.972,E2 -13747.972} C_VEL
LIN {X 0,Y 355.012,Z 223.054,A -85,B 0,C 180,E1 -13749.023,E2 -13749.023} C_VEL
LIN {X 0,Y 353.756,Z 295.503,A -85,B 0,C 180,E1 -13750.525,E2 -13750.525} C_VEL
LIN {X 0,Y 353.145,Z 308.757,A -85,B 0,C 180,E1 -13751.018,E2 -13751.018} C_VEL
LIN {X 0,Y 352.336,Z 320.946,A -85,B 0,C 180,E1 -13751.689,E2 -13751.689} C_VEL
LIN {X 0,Y 351.449,Z 332.452,A -85,B 0,C 180,E1 -13752.545,E2 -13752.545} C_VEL
LIN {X 0,Y 350.321,Z 344.256,A -85,B 0,C 180,E1 -13753.688,E2 -13753.688} C_VEL
LIN {X 0,Y 349.45,Z 354.026,A -85,B 0,C 180,E1 -13754.876,E2 -13754.876} C_VEL
LIN {X 0,Y 348.54,Z 363.532,A -85,B 0,C 180,E1 -13756.294,E2 -13756.294} C_VEL
LIN {X 0,Y 347.76,Z 371.506,A -85,B 0,C 180,E1 -13757.748,E2 -13757.748} C_VEL
LIN {X 0,Y 347.054,Z 379.275,A -85,B 0,C 180,E1 -13759.499,E2 -13759.499} C_VEL
LIN {X 0,Y 346.576,Z 385.502,A -85,B 0,C 180,E1 -13761.252,E2 -13761.252} C_VEL
LIN {X 0,Y 346.323,Z 390.436,A -85,B 0,C 180,E1 -13763.006,E2 -13763.006} C_VEL
LIN {X 0,Y 346.196,Z 393.747,A -85,B 0,C 180,E1 -13764.503,E2 -13764.503} C_VEL
LIN {X 0,Y 346.161,Z 396.959,A -85,B 0,C 180,E1 -13766.508,E2 -13766.508} C_VEL
LIN {X 0,Y 346.194,Z 399.132,A -85,B 0,C 180,E1 -13768.837,E2 -13768.837} C_VEL
LIN {X 0,Y 346.235,Z 399.588,A -85,B 0,C 180,E1 -13770,E2 -13770} C_VEL
LIN {X 0,Y 346.162,Z 399.627,A -85,B 0,C 180,E1 -13771.163,E2 -13771.163} C_VEL
LIN {X 0,Y 346.143,Z 398.55,A -85,B 0,C 180,E1 -13773.492,E2 -13773.492} C_VEL
LIN {X 0,Y 346.155,Z 397.401,A -85,B 0,C 180,E1 -13774.658,E2 -13774.658} C_VEL
LIN {X 0,Y 346.199,Z 395.726,A -85,B 0,C 180,E1 -13775.885,E2 -13775.885} C_VEL
LIN {X 0,Y 346.551,Z 391.404,A -85,B 0,C 180,E1 -13778.161,E2 -13778.161} C_VEL
LIN {X 0,Y 347.031,Z 386.835,A -85,B 0,C 180,E1 -13779.912,E2 -13779.912} C_VEL
LIN {X 0,Y 347.904,Z 379.946,A -85,B 0,C 180,E1 -13781.95,E2 -13781.95} C_VEL
LIN {X 0,Y 349.062,Z 372.507,A -85,B 0,C 180,E1 -13783.684,E2 -13783.684} C_VEL
LIN {X 0,Y 350.075,Z 364.951,A -85,B 0,C 180,E1 -13785.128,E2 -13785.128} C_VEL
LIN {X 0,Y 351.34,Z 355.832,A -85,B 0,C 180,E1 -13786.562,E2 -13786.562} C_VEL
LIN {X 0,Y 352.808,Z 345.742,A -85,B 0,C 180,E1 -13787.835,E2 -13787.835} C_VEL
LIN {X 0,Y 354.213,Z 334.581,A -85,B 0,C 180,E1 -13788.959,E2 -13788.959} C_VEL
LIN {X 0,Y 355.405,Z 324.056,A -85,B 0,C 180,E1 -13789.794,E2 -13789.794} C_VEL
LIN {X 0,Y 356.551,Z 311.447,A -85,B 0,C 180,E1 -13790.555,E2 -13790.555} C_VEL
LIN {X 0,Y 357.447,Z 299.04,A -85,B 0,C 180,E1 -13791.066,E2 -13791.066} C_VEL
LIN {X 0,Y 357.987,Z 283.584,A -85,B 0,C 180,E1 -13791.447,E2 -13791.447} C_VEL
LIN {X 0,Y 359.134,Z 223.619,A -85,B 0,C 180,E1 -13792.697,E2 -13792.697} C_VEL
LIN {X 0,Y 355.564,Z 202.272,A -85,B 0,C 180,E1 -13793.47,E2 -13793.47} C_VEL
LIN {X 0,Y 352.148,Z 186.078,A -85,B 0,C 180,E1 -13794.161,E2 -13794.161} C_VEL
LIN {X 0,Y 352.866,Z 178.473,A -85,B 0,C 180,E1 -13795.987,E2 -13795.987} C_VEL
LIN {X 0,Y 351.223,Z 169.896,A -85,B 0,C 180,E1 -13798.303,E2 -13798.303} C_VEL
LIN {X 0,Y 348.87,Z 159.542,A -85,B 0,C 180,E1 -13801.247,E2 -13801.247} C_VEL
LIN {X 0,Y 347.773,Z 155.165,A -85,B 0,C 180,E1 -13802.606,E2 -13802.606} C_VEL
LIN {X 0,Y 347.771,Z 155.165,A -85,B 0,C 180,E1 -13806.064,E2 -13806.064} C_VEL
LIN {X 0,Y 347.733,Z 155.172,A -85,B 0,C 180,E1 -13808.795,E2 -13808.795} C_VEL
LIN {X 0,Y 347.744,Z 155.164,A -85,B 0,C 180,E1 -13811.831,E2 -13811.831} C_VEL
LIN {X 0,Y 347.703,Z 155.175,A -85,B 0,C 180,E1 -13815.027,E2 -13815.027} C_VEL
LIN {X 0,Y 347.74,Z 155.17,A -85,B 0,C 180,E1 -13818.399,E2 -13818.399} C_VEL
LIN {X 0,Y 347.763,Z 155.161,A -85,B 0,C 180,E1 -13822.014,E2 -13822.014} C_VEL
LIN {X 0,Y 347.745,Z 155.161,A -85,B 0,C 180,E1 -13825.535,E2 -13825.535} C_VEL
LIN {X 0,Y 347.746,Z 155.166,A -85,B 0,C 180,E1 -13828.3,E2 -13828.3} C_VEL
LIN {X 0,Y 347.746,Z 155.167,A -85,B 0,C 180,E1 -13830.984,E2 -13830.984} C_VEL
LIN {X 0,Y 347.735,Z 155.16,A -85,B 0,C 180,E1 -13833.599,E2 -13833.599} C_VEL
LIN {X 0,Y 347.748,Z 155.166,A -85,B 0,C 180,E1 -13836.158,E2 -13836.158} C_VEL
LIN {X 0,Y 347.765,Z 155.166,A -85,B 0,C 180,E1 -13839.906,E2 -13839.906} C_VEL
LIN {X 0,Y 347.792,Z 155.158,A -85,B 0,C 180,E1 -13843.566,E2 -13843.566} C_VEL
LIN {X 0,Y 347.887,Z 155.138,A -85,B 0,C 180,E1 -13847.16,E2 -13847.16} C_VEL
LIN {X 0,Y 347.936,Z 155.138,A -85,B 0,C 180,E1 -13850.7,E2 -13850.7} C_VEL
LIN {X 0,Y 348.042,Z 155.13,A -85,B 0,C 180,E1 -13854.205,E2 -13854.205} C_VEL
LIN {X 0,Y 348.19,Z 155.104,A -85,B 0,C 180,E1 -13857.686,E2 -13857.686} C_VEL
LIN {X 0,Y 348.121,Z 155.112,A -85,B 0,C 180,E1 -13861.156,E2 -13861.156} C_VEL
LIN {X 0,Y 348.204,Z 155.106,A -85,B 0,C 180,E1 -13862.313,E2 -13862.313} C_VEL
LIN {X 0,Y 348.058,Z 155.122,A -85,B 0,C 180,E1 -13866.958,E2 -13866.958} C_VEL
LIN {X 0,Y 347.898,Z 155.139,A -85,B 0,C 180,E1 -13870.475,E2 -13870.475} C_VEL
LIN {X 0,Y 347.899,Z 155.142,A -85,B 0,C 180,E1 -13874.149,E2 -13874.149} C_VEL
LIN {X 0,Y 347.83,Z 155.151,A -85,B 0,C 180,E1 -13878.259,E2 -13878.259} C_VEL
LIN {X 0,Y 347.768,Z 155.159,A -85,B 0,C 180,E1 -13881.626,E2 -13881.626} C_VEL
LIN {X 0,Y 347.811,Z 155.158,A -85,B 0,C 180,E1 -13885.108,E2 -13885.108} C_VEL
LIN {X 0,Y 347.809,Z 155.158,A -85,B 0,C 180,E1 -13887.693,E2 -13887.693} C_VEL
LIN {X 0,Y 347.763,Z 155.166,A -85,B 0,C 180,E1 -13890.346,E2 -13890.346} C_VEL
LIN {X 0,Y 347.743,Z 155.169,A -85,B 0,C 180,E1 -13894.463,E2 -13894.463} C_VEL
LIN {X 0,Y 347.772,Z 155.169,A -85,B 0,C 180,E1 -13897.988,E2 -13897.988} C_VEL
LIN {X 0,Y 347.749,Z 155.17,A -85,B 0,C 180,E1 -13901.83,E2 -13901.83} C_VEL
LIN {X 0,Y 347.766,Z 155.217,A -85,B 0,C 180,E1 -13902.904,E2 -13902.904} C_VEL
LIN {X 0,Y 349.949,Z 164.359,A -85,B 0,C 180,E1 -13905.708,E2 -13905.708} C_VEL
LIN {X 0,Y 357.65,Z 182.011,A -85,B 0,C 180,E1 -13906.794,E2 -13906.794} C_VEL
LIN {X 0,Y 359.938,Z 191.782,A -85,B 0,C 180,E1 -13907.206,E2 -13907.206} C_VEL
LIN {X 0,Y 358.024,Z 271.814,A -85,B 0,C 180,E1 -13908.883,E2 -13908.883} C_VEL
LIN {X 0,Y 357.331,Z 285.099,A -85,B 0,C 180,E1 -13909.391,E2 -13909.391} C_VEL
LIN {X 0,Y 356.496,Z 297.506,A -85,B 0,C 180,E1 -13910.1,E2 -13910.1} C_VEL
LIN {X 0,Y 355.449,Z 308.441,A -85,B 0,C 180,E1 -13910.932,E2 -13910.932} C_VEL
LIN {X 0,Y 354.117,Z 319.679,A -85,B 0,C 180,E1 -13912.03,E2 -13912.03} C_VEL
LIN {X 0,Y 352.813,Z 329.996,A -85,B 0,C 180,E1 -13913.302,E2 -13913.302} C_VEL
LIN {X 0,Y 351.432,Z 339.506,A -85,B 0,C 180,E1 -13914.75,E2 -13914.75} C_VEL
LIN {X 0,Y 350.339,Z 347.086,A -85,B 0,C 180,E1 -13916.173,E2 -13916.173} C_VEL
LIN {X 0,Y 349.051,Z 355.13,A -85,B 0,C 180,E1 -13918.046,E2 -13918.046} C_VEL
LIN {X 0,Y 348.173,Z 360.774,A -85,B 0,C 180,E1 -13919.693,E2 -13919.693} C_VEL
LIN {X 0,Y 347.377,Z 365.949,A -85,B 0,C 180,E1 -13921.612,E2 -13921.612} C_VEL
LIN {X 0,Y 346.81,Z 369.792,A -85,B 0,C 180,E1 -13923.524,E2 -13923.524} C_VEL
LIN {X 0,Y 346.524,Z 371.664,A -85,B 0,C 180,E1 -13924.792,E2 -13924.792} C_VEL
LIN {X 0,Y 346.319,Z 373.04,A -85,B 0,C 180,E1 -13926.054,E2 -13926.054} C_VEL
LIN {X 0,Y 346.137,Z 373.97,A -85,B 0,C 180,E1 -13927.308,E2 -13927.308} C_VEL
LIN {X 0,Y 346.05,Z 374.46,A -85,B 0,C 180,E1 -13929.101,E2 -13929.101} C_VEL
LIN {X 0,Y 346.019,Z 373.956,A -85,B 0,C 180,E1 -13931.036,E2 -13931.036} C_VEL
LIN {X 0,Y 346.082,Z 372.685,A -85,B 0,C 180,E1 -13932.637,E2 -13932.637} C_VEL
LIN {X 0,Y 346.352,Z 369.933,A -85,B 0,C 180,E1 -13934.705,E2 -13934.705} C_VEL
LIN {X 0,Y 346.684,Z 366.015,A -85,B 0,C 180,E1 -13936.667,E2 -13936.667} C_VEL
LIN {X 0,Y 347.041,Z 361.659,A -85,B 0,C 180,E1 -13938.316,E2 -13938.316} C_VEL
LIN {X 0,Y 347.604,Z 355.651,A -85,B 0,C 180,E1 -13940.104,E2 -13940.104} C_VEL
LIN {X 0,Y 348.335,Z 348.15,A -85,B 0,C 180,E1 -13941.881,E2 -13941.881} C_VEL
LIN {X 0,Y 349.089,Z 340.506,A -85,B 0,C 180,E1 -13943.353,E2 -13943.353} C_VEL
LIN {X 0,Y 350.051,Z 331.22,A -85,B 0,C 180,E1 -13944.817,E2 -13944.817} C_VEL
LIN {X 0,Y 351.035,Z 320.881,A -85,B 0,C 180,E1 -13946.126,E2 -13946.126} C_VEL
LIN {X 0,Y 352.038,Z 308.796,A -85,B 0,C 180,E1 -13947.337,E2 -13947.337} C_VEL
LIN {X 0,Y 352.75,Z 297.532,A -85,B 0,C 180,E1 -13948.216,E2 -13948.216} C_VEL
LIN {X 0,Y 353.399,Z 285.151,A -85,B 0,C 180,E1 -13948.932,E2 -13948.932} C_VEL
LIN {X 0,Y 353.962,Z 272.408,A -85,B 0,C 180,E1 -13949.431,E2 -13949.431} C_VEL
LIN {X 0,Y 354.42,Z 246.752,A -85,B 0,C 180,E1 -13950,E2 -13950} C_VEL
LIN {X 0,Y 355.386,Z 188.745,A -85,B 0,C 180,E1 -13951.187,E2 -13951.187} C_VEL
LIN {X 0,Y 352.033,Z 171.371,A -85,B 0,C 180,E1 -13951.736,E2 -13951.736} C_VEL
LIN {X 0,Y 349.579,Z 163.332,A -85,B 0,C 180,E1 -13952.067,E2 -13952.067} C_VEL
LIN {X 0,Y 347.857,Z 155.153,A -85,B 0,C 180,E1 -13954.418,E2 -13954.418} C_VEL
LIN {X 0,Y 348.05,Z 155.127,A -85,B 0,C 180,E1 -13956.959,E2 -13956.959} C_VEL
LIN {X 0,Y 347.884,Z 155.148,A -85,B 0,C 180,E1 -13960.476,E2 -13960.476} C_VEL
LIN {X 0,Y 347.848,Z 155.155,A -85,B 0,C 180,E1 -13964.119,E2 -13964.119} C_VEL
LIN {X 0,Y 347.804,Z 155.158,A -85,B 0,C 180,E1 -13964.726,E2 -13964.726} C_VEL
LIN {X 0,Y 347.109,Z 155.251,A -85,B 0,C 180,E1 -13965.693,E2 -13965.693} C_VEL
LIN {X 0,Y 344.22,Z 155.607,A -85,B 0,C 180,E1 -13967.266,E2 -13967.266} C_VEL
LIN {X 0,Y 341.788,Z 155.909,A -85,B 0,C 180,E1 -13968.539,E2 -13968.539} C_VEL
LIN {X 0,Y 340.747,Z 156.042,A -85,B 0,C 180,E1 -13969.525,E2 -13969.525} C_VEL
LIN {X 0,Y 340.664,Z 156.046,A -85,B 0,C 180,E1 -13969.859,E2 -13969.859} C_VEL
LIN {X 0,Y 340.693,Z 156.046,A -85,B 0,C 180,E1 -13973.076,E2 -13973.076} C_VEL
LIN {X 0,Y 340.705,Z 156.044,A -85,B 0,C 180,E1 -13976.989,E2 -13976.989} C_VEL
LIN {X 0,Y 340.689,Z 156.047,A -85,B 0,C 180,E1 -13981.046,E2 -13981.046} C_VEL
LIN {X 0,Y 340.712,Z 156.046,A -85,B 0,C 180,E1 -13985.28,E2 -13985.28} C_VEL
LIN {X 0,Y 340.69,Z 156.044,A -85,B 0,C 180,E1 -13988.383,E2 -13988.383} C_VEL
LIN {X 0,Y 340.688,Z 156.044,A -85,B 0,C 180,E1 -13992.045,E2 -13992.045} C_VEL
LIN {X 0,Y 340.648,Z 156.05,A -85,B 0,C 180,E1 -13996.228,E2 -13996.228} C_VEL
LIN {X 0,Y 340.667,Z 156.051,A -85,B 0,C 180,E1 -13998.689,E2 -13998.689} C_VEL
LIN {X 0,Y 340.718,Z 156.04,A -85,B 0,C 180,E1 -14001.772,E2 -14001.772} C_VEL
LIN {X 0,Y 340.722,Z 156.04,A -85,B 0,C 180,E1 -14005.597,E2 -14005.597} C_VEL
LIN {X 0,Y 340.692,Z 156.046,A -85,B 0,C 180,E1 -14008.956,E2 -14008.956} C_VEL
LIN {X 0,Y 340.71,Z 156.043,A -85,B 0,C 180,E1 -14013.013,E2 -14013.013} C_VEL
LIN {X 0,Y 340.701,Z 156.044,A -85,B 0,C 180,E1 -14016.926,E2 -14016.926} C_VEL
LIN {X 0,Y 340.691,Z 156.046,A -85,B 0,C 180,E1 -14020.728,E2 -14020.728} C_VEL
LIN {X 0,Y 340.728,Z 156.039,A -85,B 0,C 180,E1 -14023.216,E2 -14023.216} C_VEL
LIN {X 0,Y 340.817,Z 156.029,A -85,B 0,C 180,E1 -14026.89,E2 -14026.89} C_VEL
LIN {X 0,Y 340.883,Z 156.022,A -85,B 0,C 180,E1 -14030.507,E2 -14030.507} C_VEL
LIN {X 0,Y 341.012,Z 156.004,A -85,B 0,C 180,E1 -14032.898,E2 -14032.898} C_VEL
LIN {X 0,Y 340.811,Z 156.029,A -85,B 0,C 180,E1 -14035.269,E2 -14035.269} C_VEL
LIN {X 0,Y 341.121,Z 155.994,A -85,B 0,C 180,E1 -14037.639,E2 -14037.639} C_VEL
LIN {X 0,Y 341.092,Z 155.995,A -85,B 0,C 180,E1 -14041.181,E2 -14041.181} C_VEL
LIN {X 0,Y 341.128,Z 155.99,A -85,B 0,C 180,E1 -14042.362,E2 -14042.362} C_VEL
LIN {X 0,Y 341.004,Z 156.006,A -85,B 0,C 180,E1 -14047.104,E2 -14047.104} C_VEL
LIN {X 0,Y 340.851,Z 156.024,A -85,B 0,C 180,E1 -14050.695,E2 -14050.695} C_VEL
LIN {X 0,Y 340.823,Z 156.027,A -85,B 0,C 180,E1 -14054.327,E2 -14054.327} C_VEL
LIN {X 0,Y 340.761,Z 156.035,A -85,B 0,C 180,E1 -14058.426,E2 -14058.426} C_VEL
LIN {X 0,Y 340.723,Z 156.041,A -85,B 0,C 180,E1 -14061.842,E2 -14061.842} C_VEL
LIN {X 0,Y 340.719,Z 156.042,A -85,B 0,C 180,E1 -14065.669,E2 -14065.669} C_VEL
LIN {X 0,Y 340.707,Z 156.043,A -85,B 0,C 180,E1 -14069.675,E2 -14069.675} C_VEL
LIN {X 0,Y 340.689,Z 156.045,A -85,B 0,C 180,E1 -14072.436,E2 -14072.436} C_VEL
LIN {X 0,Y 340.72,Z 156.043,A -85,B 0,C 180,E1 -14075.279,E2 -14075.279} C_VEL
LIN {X 0,Y 340.698,Z 156.045,A -85,B 0,C 180,E1 -14078.383,E2 -14078.383} C_VEL
LIN {X 0,Y 340.697,Z 156.043,A -85,B 0,C 180,E1 -14082.044,E2 -14082.044} C_VEL
LIN {X 0,Y 340.654,Z 156.05,A -85,B 0,C 180,E1 -14086.227,E2 -14086.227} C_VEL
LIN {X 0,Y 340.674,Z 156.051,A -85,B 0,C 180,E1 -14088.688,E2 -14088.688} C_VEL
LIN {X 0,Y 340.723,Z 156.04,A -85,B 0,C 180,E1 -14091.771,E2 -14091.771} C_VEL
LIN {X 0,Y 340.727,Z 156.04,A -85,B 0,C 180,E1 -14095.595,E2 -14095.595} C_VEL
LIN {X 0,Y 340.755,Z 156.041,A -85,B 0,C 180,E1 -14099.923,E2 -14099.923} C_VEL
LIN {X 0,Y 343.242,Z 168.576,A -85,B 0,C 180,E1 -14103.227,E2 -14103.227} C_VEL
LIN {X 0,Y 344.255,Z 175.376,A -85,B 0,C 180,E1 -14104.937,E2 -14104.937} C_VEL
LIN {X 0,Y 343.05,Z 186.795,A -85,B 0,C 180,E1 -14107.608,E2 -14107.608} C_VEL
LIN {X 0,Y 348.225,Z 223.682,A -85,B 0,C 180,E1 -14108.698,E2 -14108.698} C_VEL
LIN {X 0,Y 346.937,Z 295.018,A -85,B 0,C 180,E1 -14110.203,E2 -14110.203} C_VEL
LIN {X 0,Y 346.307,Z 308.349,A -85,B 0,C 180,E1 -14110.706,E2 -14110.706} C_VEL
LIN {X 0,Y 345.382,Z 321.703,A -85,B 0,C 180,E1 -14111.461,E2 -14111.461} C_VEL
LIN {X 0,Y 344.476,Z 332.926,A -85,B 0,C 180,E1 -14112.333,E2 -14112.333} C_VEL
LIN {X 0,Y 343.333,Z 344.586,A -85,B 0,C 180,E1 -14113.499,E2 -14113.499} C_VEL
LIN {X 0,Y 342.418,Z 354.348,A -85,B 0,C 180,E1 -14114.724,E2 -14114.724} C_VEL
LIN {X 0,Y 341.616,Z 362.782,A -85,B 0,C 180,E1 -14116.011,E2 -14116.011} C_VEL
LIN {X 0,Y 340.786,Z 370.838,A -85,B 0,C 180,E1 -14117.494,E2 -14117.494} C_VEL
LIN {X 0,Y 340.012,Z 378.706,A -85,B 0,C 180,E1 -14119.279,E2 -14119.279} C_VEL
LIN {X 0,Y 339.522,Z 384.994,A -85,B 0,C 180,E1 -14121.069,E2 -14121.069} C_VEL
LIN {X 0,Y 339.25,Z 389.981,A -85,B 0,C 180,E1 -14122.86,E2 -14122.86} C_VEL
LIN {X 0,Y 339.098,Z 393.671,A -85,B 0,C 180,E1 -14124.57,E2 -14124.57} C_VEL
LIN {X 0,Y 339.086,Z 396.601,A -85,B 0,C 180,E1 -14126.435,E2 -14126.435} C_VEL
LIN {X 0,Y 339.096,Z 398.818,A -85,B 0,C 180,E1 -14128.812,E2 -14128.812} C_VEL
LIN {X 0,Y 339.14,Z 399.316,A -85,B 0,C 180,E1 -14130,E2 -14130} C_VEL
LIN {X 0,Y 339.063,Z 399.376,A -85,B 0,C 180,E1 -14131.187,E2 -14131.187} C_VEL
LIN {X 0,Y 339.066,Z 398.342,A -85,B 0,C 180,E1 -14133.565,E2 -14133.565} C_VEL
LIN {X 0,Y 339.059,Z 397.232,A -85,B 0,C 180,E1 -14134.756,E2 -14134.756} C_VEL
LIN {X 0,Y 339.132,Z 395.675,A -85,B 0,C 180,E1 -14135.947,E2 -14135.947} C_VEL
LIN {X 0,Y 339.356,Z 392.566,A -85,B 0,C 180,E1 -14137.736,E2 -14137.736} C_VEL
LIN {X 0,Y 339.818,Z 388.415,A -85,B 0,C 180,E1 -14139.523,E2 -14139.523} C_VEL
LIN {X 0,Y 340.592,Z 382.099,A -85,B 0,C 180,E1 -14141.606,E2 -14141.606} C_VEL
LIN {X 0,Y 341.765,Z 375.25,A -85,B 0,C 180,E1 -14143.376,E2 -14143.376} C_VEL
LIN {X 0,Y 343.037,Z 366.742,A -85,B 0,C 180,E1 -14145.142,E2 -14145.142} C_VEL
LIN {X 0,Y 344.251,Z 358.03,A -85,B 0,C 180,E1 -14146.607,E2 -14146.607} C_VEL
LIN {X 0,Y 345.876,Z 347.331,A -85,B 0,C 180,E1 -14148.051,E2 -14148.051} C_VEL
LIN {X 0,Y 347.316,Z 336.703,A -85,B 0,C 180,E1 -14149.197,E2 -14149.197} C_VEL
LIN {X 0,Y 348.763,Z 324.833,A -85,B 0,C 180,E1 -14150.187,E2 -14150.187} C_VEL
LIN {X 0,Y 349.963,Z 312.539,A -85,B 0,C 180,E1 -14150.96,E2 -14150.96} C_VEL
LIN {X 0,Y 350.941,Z 299.949,A -85,B 0,C 180,E1 -14151.514,E2 -14151.514} C_VEL
LIN {X 0,Y 351.542,Z 285.287,A -85,B 0,C 180,E1 -14151.899,E2 -14151.899} C_VEL
LIN {X 0,Y 352.801,Z 224.603,A -85,B 0,C 180,E1 -14153.189,E2 -14153.189} C_VEL
LIN {X 0,Y 349.271,Z 203.551,A -85,B 0,C 180,E1 -14153.982,E2 -14153.982} C_VEL
LIN {X 0,Y 345.491,Z 185.839,A -85,B 0,C 180,E1 -14154.752,E2 -14154.752} C_VEL
LIN {X 0,Y 346.053,Z 181.161,A -85,B 0,C 180,E1 -14155.89,E2 -14155.89} C_VEL
LIN {X 0,Y 345.332,Z 176.099,A -85,B 0,C 180,E1 -14157.251,E2 -14157.251} C_VEL
LIN {X 0,Y 342.812,Z 164.491,A -85,B 0,C 180,E1 -14160.565,E2 -14160.565} C_VEL
LIN {X 0,Y 340.714,Z 156.048,A -85,B 0,C 180,E1 -14163.135,E2 -14163.135} C_VEL
LIN {X 0,Y 340.704,Z 156.04,A -85,B 0,C 180,E1 -14166.742,E2 -14166.742} C_VEL
LIN {X 0,Y 340.653,Z 156.045,A -85,B 0,C 180,E1 -14170.239,E2 -14170.239} C_VEL
LIN {X 0,Y 340.675,Z 156.052,A -85,B 0,C 180,E1 -14172.905,E2 -14172.905} C_VEL
LIN {X 0,Y 340.674,Z 156.048,A -85,B 0,C 180,E1 -14177.095,E2 -14177.095} C_VEL
LIN {X 0,Y 340.657,Z 156.05,A -85,B 0,C 180,E1 -14180.241,E2 -14180.241} C_VEL
LIN {X 0,Y 340.708,Z 156.045,A -85,B 0,C 180,E1 -14183.56,E2 -14183.56} C_VEL
LIN {X 0,Y 340.694,Z 156.04,A -85,B 0,C 180,E1 -14186.153,E2 -14186.153} C_VEL
LIN {X 0,Y 340.721,Z 156.036,A -85,B 0,C 180,E1 -14190.035,E2 -14190.035} C_VEL
LIN {X 0,Y 340.712,Z 156.034,A -85,B 0,C 180,E1 -14193.011,E2 -14193.011} C_VEL
LIN {X 0,Y 340.716,Z 156.041,A -85,B 0,C 180,E1 -14195.635,E2 -14195.635} C_VEL
LIN {X 0,Y 340.706,Z 156.043,A -85,B 0,C 180,E1 -14199.471,E2 -14199.471} C_VEL
LIN {X 0,Y 340.759,Z 156.029,A -85,B 0,C 180,E1 -14201.978,E2 -14201.978} C_VEL
LIN {X 0,Y 340.834,Z 156.026,A -85,B 0,C 180,E1 -14205.729,E2 -14205.729} C_VEL
LIN {X 0,Y 340.847,Z 156.026,A -85,B 0,C 180,E1 -14209.305,E2 -14209.305} C_VEL
LIN {X 0,Y 341.004,Z 156.001,A -85,B 0,C 180,E1 -14212.896,E2 -14212.896} C_VEL
LIN {X 0,Y 340.816,Z 156.029,A -85,B 0,C 180,E1 -14215.268,E2 -14215.268} C_VEL
LIN {X 0,Y 341.127,Z 155.983,A -85,B 0,C 180,E1 -14217.638,E2 -14217.638} C_VEL
LIN {X 0,Y 341.092,Z 155.987,A -85,B 0,C 180,E1 -14221.18,E2 -14221.18} C_VEL
LIN {X 0,Y 341.165,Z 155.983,A -85,B 0,C 180,E1 -14222.361,E2 -14222.361} C_VEL
LIN {X 0,Y 341.005,Z 156.002,A -85,B 0,C 180,E1 -14227.103,E2 -14227.103} C_VEL
LIN {X 0,Y 340.85,Z 156.017,A -85,B 0,C 180,E1 -14230.694,E2 -14230.694} C_VEL
LIN {X 0,Y 340.864,Z 156.018,A -85,B 0,C 180,E1 -14234.324,E2 -14234.324} C_VEL
LIN {X 0,Y 340.787,Z 156.028,A -85,B 0,C 180,E1 -14238.44,E2 -14238.44} C_VEL
LIN {X 0,Y 340.718,Z 156.037,A -85,B 0,C 180,E1 -14241.841,E2 -14241.841} C_VEL
LIN {X 0,Y 340.771,Z 156.037,A -85,B 0,C 180,E1 -14245.664,E2 -14245.664} C_VEL
LIN {X 0,Y 340.74,Z 156.039,A -85,B 0,C 180,E1 -14248.319,E2 -14248.319} C_VEL
LIN {X 0,Y 340.703,Z 156.046,A -85,B 0,C 180,E1 -14251.043,E2 -14251.043} C_VEL
LIN {X 0,Y 340.717,Z 156.046,A -85,B 0,C 180,E1 -14255.278,E2 -14255.278} C_VEL
LIN {X 0,Y 340.708,Z 156.045,A -85,B 0,C 180,E1 -14258.385,E2 -14258.385} C_VEL
LIN {X 0,Y 340.73,Z 156.108,A -85,B 0,C 180,E1 -14262.354,E2 -14262.354} C_VEL
LIN {X 0,Y 342.735,Z 164.417,A -85,B 0,C 180,E1 -14265.026,E2 -14265.026} C_VEL
LIN {X 0,Y 351.529,Z 184.233,A -85,B 0,C 180,E1 -14266.316,E2 -14266.316} C_VEL
LIN {X 0,Y 353.568,Z 192.56,A -85,B 0,C 180,E1 -14266.687,E2 -14266.687} C_VEL
LIN {X 0,Y 351.666,Z 271.193,A -85,B 0,C 180,E1 -14268.365,E2 -14268.365} C_VEL
LIN {X 0,Y 350.949,Z 284.428,A -85,B 0,C 180,E1 -14268.865,E2 -14268.865} C_VEL
LIN {X 0,Y 350.054,Z 297.366,A -85,B 0,C 180,E1 -14269.606,E2 -14269.606} C_VEL
LIN {X 0,Y 348.972,Z 308.24,A -85,B 0,C 180,E1 -14270.439,E2 -14270.439} C_VEL
LIN {X 0,Y 347.625,Z 319.177,A -85,B 0,C 180,E1 -14271.51,E2 -14271.51} C_VEL
LIN {X 0,Y 346.201,Z 329.952,A -85,B 0,C 180,E1 -14272.848,E2 -14272.848} C_VEL
LIN {X 0,Y 344.726,Z 339.557,A -85,B 0,C 180,E1 -14274.327,E2 -14274.327} C_VEL
LIN {X 0,Y 343.555,Z 347.137,A -85,B 0,C 180,E1 -14275.767,E2 -14275.767} C_VEL
LIN {X 0,Y 342.489,Z 353.721,A -85,B 0,C 180,E1 -14277.28,E2 -14277.28} C_VEL
LIN {X 0,Y 341.418,Z 359.922,A -85,B 0,C 180,E1 -14279.028,E2 -14279.028} C_VEL
LIN {X 0,Y 340.549,Z 365.343,A -85,B 0,C 180,E1 -14280.989,E2 -14280.989} C_VEL
LIN {X 0,Y 339.871,Z 369.41,A -85,B 0,C 180,E1 -14282.94,E2 -14282.94} C_VEL
LIN {X 0,Y 339.552,Z 371.457,A -85,B 0,C 180,E1 -14284.237,E2 -14284.237} C_VEL
LIN {X 0,Y 339.274,Z 373.133,A -85,B 0,C 180,E1 -14285.705,E2 -14285.705} C_VEL
LIN {X 0,Y 338.978,Z 374.596,A -85,B 0,C 180,E1 -14288.087,E2 -14288.087} C_VEL
LIN {X 0,Y 338.95,Z 374.701,A -85,B 0,C 180,E1 -14289.36,E2 -14289.36} C_VEL
LIN {X 0,Y 338.908,Z 374.367,A -85,B 0,C 180,E1 -14290.622,E2 -14290.622} C_VEL
LIN {X 0,Y 338.989,Z 373.061,A -85,B 0,C 180,E1 -14292.491,E2 -14292.491} C_VEL
LIN {X 0,Y 339.317,Z 369.723,A -85,B 0,C 180,E1 -14294.995,E2 -14294.995} C_VEL
LIN {X 0,Y 339.64,Z 365.989,A -85,B 0,C 180,E1 -14296.843,E2 -14296.843} C_VEL
LIN {X 0,Y 340.04,Z 361.1,A -85,B 0,C 180,E1 -14298.677,E2 -14298.677} C_VEL
LIN {X 0,Y 340.604,Z 354.912,A -85,B 0,C 180,E1 -14300.499,E2 -14300.499} C_VEL
LIN {X 0,Y 341.409,Z 347.197,A -85,B 0,C 180,E1 -14302.311,E2 -14302.311} C_VEL
LIN {X 0,Y 342.281,Z 339.279,A -85,B 0,C 180,E1 -14303.812,E2 -14303.812} C_VEL
LIN {X 0,Y 343.253,Z 329.602,A -85,B 0,C 180,E1 -14305.302,E2 -14305.302} C_VEL
LIN {X 0,Y 344.322,Z 319.074,A -85,B 0,C 180,E1 -14306.607,E2 -14306.607} C_VEL
LIN {X 0,Y 345.202,Z 308.431,A -85,B 0,C 180,E1 -14307.667,E2 -14307.667} C_VEL
LIN {X 0,Y 345.973,Z 296.103,A -85,B 0,C 180,E1 -14308.618,E2 -14308.618} C_VEL
LIN {X 0,Y 346.658,Z 283.082,A -85,B 0,C 180,E1 -14309.347,E2 -14309.347} C_VEL
LIN {X 0,Y 347.216,Z 270.292,A -85,B 0,C 180,E1 -14309.819,E2 -14309.819} C_VEL
LIN {X 0,Y 348.62,Z 189.787,A -85,B 0,C 180,E1 -14311.517,E2 -14311.517} C_VEL
LIN {X 0,Y 345.467,Z 173.383,A -85,B 0,C 180,E1 -14312.048,E2 -14312.048} C_VEL
LIN {X 0,Y 342.465,Z 163.565,A -85,B 0,C 180,E1 -14312.463,E2 -14312.463} C_VEL
LIN {X 0,Y 340.808,Z 156.03,A -85,B 0,C 180,E1 -14314.658,E2 -14314.658} C_VEL
LIN {X 0,Y 340.997,Z 156.006,A -85,B 0,C 180,E1 -14317.104,E2 -14317.104} C_VEL
LIN {X 0,Y 340.836,Z 156.026,A -85,B 0,C 180,E1 -14320.695,E2 -14320.695} C_VEL
LIN {X 0,Y 340.807,Z 156.03,A -85,B 0,C 180,E1 -14324.328,E2 -14324.328} C_VEL
LIN {X 0,Y 340.746,Z 156.037,A -85,B 0,C 180,E1 -14328.423,E2 -14328.423} C_VEL
LIN {X 0,Y 340.664,Z 156.046,A -85,B 0,C 180,E1 -14329.859,E2 -14329.859} C_VEL
LIN {X 0,Y 340.016,Z 156.129,A -85,B 0,C 180,E1 -14330.845,E2 -14330.845} C_VEL
LIN {X 0,Y 337.218,Z 156.482,A -85,B 0,C 180,E1 -14332.451,E2 -14332.451} C_VEL
LIN {X 0,Y 334.82,Z 156.782,A -85,B 0,C 180,E1 -14333.75,E2 -14333.75} C_VEL
LIN {X 0,Y 333.755,Z 156.911,A -85,B 0,C 180,E1 -14334.755,E2 -14334.755} C_VEL
LIN {X 0,Y 333.65,Z 156.921,A -85,B 0,C 180,E1 -14335.096,E2 -14335.096} C_VEL
LIN {X 0,Y 333.625,Z 156.926,A -85,B 0,C 180,E1 -14338.981,E2 -14338.981} C_VEL
LIN {X 0,Y 333.641,Z 156.923,A -85,B 0,C 180,E1 -14342.588,E2 -14342.588} C_VEL
LIN {X 0,Y 333.67,Z 156.917,A -85,B 0,C 180,E1 -14346.14,E2 -14346.14} C_VEL
LIN {X 0,Y 333.617,Z 156.93,A -85,B 0,C 180,E1 -14349.197,E2 -14349.197} C_VEL
LIN {X 0,Y 333.624,Z 156.925,A -85,B 0,C 180,E1 -14352.5,E2 -14352.5} C_VEL
LIN {X 0,Y 333.592,Z 156.927,A -85,B 0,C 180,E1 -14355.955,E2 -14355.955} C_VEL
LIN {X 0,Y 333.601,Z 156.928,A -85,B 0,C 180,E1 -14359.326,E2 -14359.326} C_VEL
LIN {X 0,Y 333.661,Z 156.922,A -85,B 0,C 180,E1 -14363.17,E2 -14363.17} C_VEL
LIN {X 0,Y 333.672,Z 156.919,A -85,B 0,C 180,E1 -14365.342,E2 -14365.342} C_VEL
LIN {X 0,Y 333.629,Z 156.925,A -85,B 0,C 180,E1 -14368.223,E2 -14368.223} C_VEL
LIN {X 0,Y 333.629,Z 156.924,A -85,B 0,C 180,E1 -14371.021,E2 -14371.021} C_VEL
LIN {X 0,Y 333.657,Z 156.922,A -85,B 0,C 180,E1 -14374.924,E2 -14374.924} C_VEL
LIN {X 0,Y 333.64,Z 156.923,A -85,B 0,C 180,E1 -14379.017,E2 -14379.017} C_VEL
LIN {X 0,Y 333.707,Z 156.914,A -85,B 0,C 180,E1 -14381.585,E2 -14381.585} C_VEL
LIN {X 0,Y 333.761,Z 156.908,A -85,B 0,C 180,E1 -14385.611,E2 -14385.611} C_VEL
LIN {X 0,Y 333.812,Z 156.901,A -85,B 0,C 180,E1 -14389.078,E2 -14389.078} C_VEL
LIN {X 0,Y 333.966,Z 156.882,A -85,B 0,C 180,E1 -14392.747,E2 -14392.747} C_VEL
LIN {X 0,Y 333.778,Z 156.905,A -85,B 0,C 180,E1 -14395.169,E2 -14395.169} C_VEL
LIN {X 0,Y 334.062,Z 156.873,A -85,B 0,C 180,E1 -14397.589,E2 -14397.589} C_VEL
LIN {X 0,Y 334.062,Z 156.87,A -85,B 0,C 180,E1 -14401.206,E2 -14401.206} C_VEL
LIN {X 0,Y 334.068,Z 156.87,A -85,B 0,C 180,E1 -14402.412,E2 -14402.412} C_VEL
LIN {X 0,Y 333.989,Z 156.881,A -85,B 0,C 180,E1 -14406.04,E2 -14406.04} C_VEL
LIN {X 0,Y 333.917,Z 156.887,A -85,B 0,C 180,E1 -14408.473,E2 -14408.473} C_VEL
LIN {X 0,Y 333.794,Z 156.904,A -85,B 0,C 180,E1 -14412.155,E2 -14412.155} C_VEL
LIN {X 0,Y 333.722,Z 156.913,A -85,B 0,C 180,E1 -14415.89,E2 -14415.89} C_VEL
LIN {X 0,Y 333.7,Z 156.915,A -85,B 0,C 180,E1 -14418.604,E2 -14418.604} C_VEL
LIN {X 0,Y 333.655,Z 156.92,A -85,B 0,C 180,E1 -14422.281,E2 -14422.281} C_VEL
LIN {X 0,Y 333.692,Z 156.92,A -85,B 0,C 180,E1 -14425.089,E2 -14425.089} C_VEL
LIN {X 0,Y 333.654,Z 156.925,A -85,B 0,C 180,E1 -14428.978,E2 -14428.978} C_VEL
LIN {X 0,Y 333.647,Z 156.923,A -85,B 0,C 180,E1 -14432.587,E2 -14432.587} C_VEL
LIN {X 0,Y 333.678,Z 156.918,A -85,B 0,C 180,E1 -14436.139,E2 -14436.139} C_VEL
LIN {X 0,Y 333.624,Z 156.927,A -85,B 0,C 180,E1 -14439.196,E2 -14439.196} C_VEL
LIN {X 0,Y 333.633,Z 156.927,A -85,B 0,C 180,E1 -14442.499,E2 -14442.499} C_VEL
LIN {X 0,Y 333.598,Z 156.928,A -85,B 0,C 180,E1 -14445.954,E2 -14445.954} C_VEL
LIN {X 0,Y 333.606,Z 156.927,A -85,B 0,C 180,E1 -14449.325,E2 -14449.325} C_VEL
LIN {X 0,Y 333.667,Z 156.92,A -85,B 0,C 180,E1 -14453.168,E2 -14453.168} C_VEL
LIN {X 0,Y 333.678,Z 156.918,A -85,B 0,C 180,E1 -14455.341,E2 -14455.341} C_VEL
LIN {X 0,Y 333.725,Z 157.009,A -85,B 0,C 180,E1 -14459.687,E2 -14459.687} C_VEL
LIN {X 0,Y 336.132,Z 169.216,A -85,B 0,C 180,E1 -14462.945,E2 -14462.945} C_VEL
LIN {X 0,Y 337.286,Z 176.056,A -85,B 0,C 180,E1 -14464.712,E2 -14464.712} C_VEL
LIN {X 0,Y 336.12,Z 186.562,A -85,B 0,C 180,E1 -14467.222,E2 -14467.222} C_VEL
LIN {X 0,Y 341.442,Z 224.837,A -85,B 0,C 180,E1 -14468.371,E2 -14468.371} C_VEL
LIN {X 0,Y 340.093,Z 295.686,A -85,B 0,C 180,E1 -14469.906,E2 -14469.906} C_VEL
LIN {X 0,Y 339.404,Z 309.472,A -85,B 0,C 180,E1 -14470.455,E2 -14470.455} C_VEL
LIN {X 0,Y 338.436,Z 322.377,A -85,B 0,C 180,E1 -14471.223,E2 -14471.223} C_VEL
LIN {X 0,Y 337.337,Z 334.978,A -85,B 0,C 180,E1 -14472.26,E2 -14472.26} C_VEL
LIN {X 0,Y 336.223,Z 346.22,A -85,B 0,C 180,E1 -14473.453,E2 -14473.453} C_VEL
LIN {X 0,Y 335.29,Z 356.142,A -85,B 0,C 180,E1 -14474.781,E2 -14474.781} C_VEL
LIN {X 0,Y 334.283,Z 365.468,A -85,B 0,C 180,E1 -14476.318,E2 -14476.318} C_VEL
LIN {X 0,Y 333.344,Z 374.376,A -85,B 0,C 180,E1 -14478.137,E2 -14478.137} C_VEL
LIN {X 0,Y 332.728,Z 381.489,A -85,B 0,C 180,E1 -14479.964,E2 -14479.964} C_VEL
LIN {X 0,Y 332.254,Z 387.976,A -85,B 0,C 180,E1 -14482.097,E2 -14482.097} C_VEL
LIN {X 0,Y 332.034,Z 392.744,A -85,B 0,C 180,E1 -14484.174,E2 -14484.174} C_VEL
LIN {X 0,Y 332.012,Z 396.244,A -85,B 0,C 180,E1 -14486.359,E2 -14486.359} C_VEL
LIN {X 0,Y 331.999,Z 398.503,A -85,B 0,C 180,E1 -14488.787,E2 -14488.787} C_VEL
LIN {X 0,Y 332.044,Z 399.036,A -85,B 0,C 180,E1 -14490,E2 -14490} C_VEL
LIN {X 0,Y 331.966,Z 399.126,A -85,B 0,C 180,E1 -14491.213,E2 -14491.213} C_VEL
LIN {X 0,Y 331.991,Z 398.134,A -85,B 0,C 180,E1 -14493.641,E2 -14493.641} C_VEL
LIN {X 0,Y 332.006,Z 395.945,A -85,B 0,C 180,E1 -14495.779,E2 -14495.779} C_VEL
LIN {X 0,Y 332.307,Z 392.468,A -85,B 0,C 180,E1 -14497.901,E2 -14497.901} C_VEL
LIN {X 0,Y 332.793,Z 388.366,A -85,B 0,C 180,E1 -14499.726,E2 -14499.726} C_VEL
LIN {X 0,Y 333.614,Z 382.103,A -85,B 0,C 180,E1 -14501.853,E2 -14501.853} C_VEL
LIN {X 0,Y 334.832,Z 375.312,A -85,B 0,C 180,E1 -14503.658,E2 -14503.658} C_VEL
LIN {X 0,Y 336.162,Z 366.907,A -85,B 0,C 180,E1 -14505.459,E2 -14505.459} C_VEL
LIN {X 0,Y 337.466,Z 358.29,A -85,B 0,C 180,E1 -14506.951,E2 -14506.951} C_VEL
LIN {X 0,Y 339.147,Z 347.722,A -85,B 0,C 180,E1 -14508.422,E2 -14508.422} C_VEL
LIN {X 0,Y 340.663,Z 337.266,A -85,B 0,C 180,E1 -14509.587,E2 -14509.587} C_VEL
LIN {X 0,Y 342.165,Z 325.736,A -85,B 0,C 180,E1 -14510.594,E2 -14510.594} C_VEL
LIN {X 0,Y 343.398,Z 313.832,A -85,B 0,C 180,E1 -14511.38,E2 -14511.38} C_VEL
LIN {X 0,Y 344.47,Z 301.005,A -85,B 0,C 180,E1 -14511.978,E2 -14511.978} C_VEL
LIN {X 0,Y 345.107,Z 287.568,A -85,B 0,C 180,E1 -14512.369,E2 -14512.369} C_VEL
LIN {X 0,Y 346.422,Z 224.99,A -85,B 0,C 180,E1 -14513.727,E2 -14513.727} C_VEL
LIN {X 0,Y 342.967,Z 204.439,A -85,B 0,C 180,E1 -14514.525,E2 -14514.525} C_VEL
LIN {X 0,Y 338.889,Z 185.495,A -85,B 0,C 180,E1 -14515.393,E2 -14515.393} C_VEL
LIN {X 0,Y 339.173,Z 181.691,A -85,B 0,C 180,E1 -14516.356,E2 -14516.356} C_VEL
LIN {X 0,Y 336.861,Z 169.892,A -85,B 0,C 180,E1 -14519.729,E2 -14519.729} C_VEL
LIN {X 0,Y 334.42,Z 159.905,A -85,B 0,C 180,E1 -14522.794,E2 -14522.794} C_VEL
LIN {X 0,Y 333.675,Z 156.918,A -85,B 0,C 180,E1 -14523.747,E2 -14523.747} C_VEL
LIN {X 0,Y 333.665,Z 156.916,A -85,B 0,C 180,E1 -14526.831,E2 -14526.831} C_VEL
LIN {X 0,Y 333.605,Z 156.919,A -85,B 0,C 180,E1 -14530.774,E2 -14530.774} C_VEL
LIN {X 0,Y 333.592,Z 156.928,A -85,B 0,C 180,E1 -14534.249,E2 -14534.249} C_VEL
LIN {X 0,Y 333.637,Z 156.927,A -85,B 0,C 180,E1 -14537.617,E2 -14537.617} C_VEL
LIN {X 0,Y 333.636,Z 156.924,A -85,B 0,C 180,E1 -14541.206,E2 -14541.206} C_VEL
LIN {X 0,Y 333.675,Z 156.92,A -85,B 0,C 180,E1 -14543.86,E2 -14543.86} C_VEL
LIN {X 0,Y 333.646,Z 156.923,A -85,B 0,C 180,E1 -14547.413,E2 -14547.413} C_VEL
LIN {X 0,Y 333.652,Z 156.923,A -85,B 0,C 180,E1 -14551.022,E2 -14551.022} C_VEL
LIN {X 0,Y 333.665,Z 156.92,A -85,B 0,C 180,E1 -14555.085,E2 -14555.085} C_VEL
LIN {X 0,Y 333.643,Z 156.923,A -85,B 0,C 180,E1 -14559.016,E2 -14559.016} C_VEL
LIN {X 0,Y 333.711,Z 156.908,A -85,B 0,C 180,E1 -14561.584,E2 -14561.584} C_VEL
LIN {X 0,Y 333.776,Z 156.907,A -85,B 0,C 180,E1 -14565.6,E2 -14565.6} C_VEL
LIN {X 0,Y 333.817,Z 156.901,A -85,B 0,C 180,E1 -14569.077,E2 -14569.077} C_VEL
LIN {X 0,Y 333.959,Z 156.879,A -85,B 0,C 180,E1 -14572.745,E2 -14572.745} C_VEL
LIN {X 0,Y 333.782,Z 156.905,A -85,B 0,C 180,E1 -14575.168,E2 -14575.168} C_VEL
LIN {X 0,Y 334.068,Z 156.862,A -85,B 0,C 180,E1 -14577.588,E2 -14577.588} C_VEL
LIN {X 0,Y 334.063,Z 156.862,A -85,B 0,C 180,E1 -14581.205,E2 -14581.205} C_VEL
LIN {X 0,Y 334.102,Z 156.862,A -85,B 0,C 180,E1 -14582.411,E2 -14582.411} C_VEL
LIN {X 0,Y 333.963,Z 156.875,A -85,B 0,C 180,E1 -14586.493,E2 -14586.493} C_VEL
LIN {X 0,Y 333.822,Z 156.895,A -85,B 0,C 180,E1 -14589.696,E2 -14589.696} C_VEL
LIN {X 0,Y 333.798,Z 156.903,A -85,B 0,C 180,E1 -14593.391,E2 -14593.391} C_VEL
LIN {X 0,Y 333.72,Z 156.915,A -85,B 0,C 180,E1 -14597.147,E2 -14597.147} C_VEL
LIN {X 0,Y 333.718,Z 156.916,A -85,B 0,C 180,E1 -14599.691,E2 -14599.691} C_VEL
LIN {X 0,Y 333.669,Z 156.923,A -85,B 0,C 180,E1 -14603.589,E2 -14603.589} C_VEL
LIN {X 0,Y 333.735,Z 156.914,A -85,B 0,C 180,E1 -14606.246,E2 -14606.246} C_VEL
LIN {X 0,Y 333.71,Z 156.919,A -85,B 0,C 180,E1 -14608.971,E2 -14608.971} C_VEL
LIN {X 0,Y 333.642,Z 156.924,A -85,B 0,C 180,E1 -14612.586,E2 -14612.586} C_VEL
LIN {X 0,Y 333.675,Z 156.925,A -85,B 0,C 180,E1 -14616.138,E2 -14616.138} C_VEL
LIN {X 0,Y 333.645,Z 156.922,A -85,B 0,C 180,E1 -14619.192,E2 -14619.192} C_VEL
LIN {X 0,Y 333.672,Z 157.025,A -85,B 0,C 180,E1 -14621.766,E2 -14621.766} C_VEL
LIN {X 0,Y 335.578,Z 164.736,A -85,B 0,C 180,E1 -14624.338,E2 -14624.338} C_VEL
LIN {X 0,Y 345.103,Z 185.702,A -85,B 0,C 180,E1 -14625.773,E2 -14625.773} C_VEL
LIN {X 0,Y 346.768,Z 191.164,A -85,B 0,C 180,E1 -14626.055,E2 -14626.055} C_VEL
LIN {X 0,Y 347.347,Z 194.803,A -85,B 0,C 180,E1 -14626.193,E2 -14626.193} C_VEL
LIN {X 0,Y 345.29,Z 272.295,A -85,B 0,C 180,E1 -14627.877,E2 -14627.877} C_VEL
LIN {X 0,Y 344.519,Z 285.543,A -85,B 0,C 180,E1 -14628.399,E2 -14628.399} C_VEL
LIN {X 0,Y 343.608,Z 297.746,A -85,B 0,C 180,E1 -14629.117,E2 -14629.117} C_VEL
LIN {X 0,Y 342.309,Z 309.954,A -85,B 0,C 180,E1 -14630.089,E2 -14630.089} C_VEL
LIN {X 0,Y 340.863,Z 321.138,A -85,B 0,C 180,E1 -14631.243,E2 -14631.243} C_VEL
LIN {X 0,Y 339.454,Z 331.148,A -85,B 0,C 180,E1 -14632.542,E2 -14632.542} C_VEL
LIN {X 0,Y 337.893,Z 340.56,A -85,B 0,C 180,E1 -14634.051,E2 -14634.051} C_VEL
LIN {X 0,Y 336.541,Z 348.708,A -85,B 0,C 180,E1 -14635.678,E2 -14635.678} C_VEL
LIN {X 0,Y 335.142,Z 356.721,A -85,B 0,C 180,E1 -14637.674,E2 -14637.674} C_VEL
LIN {X 0,Y 334.035,Z 362.96,A -85,B 0,C 180,E1 -14639.672,E2 -14639.672} C_VEL
LIN {X 0,Y 333.216,Z 367.712,A -85,B 0,C 180,E1 -14641.669,E2 -14641.669} C_VEL
LIN {X 0,Y 332.609,Z 371.183,A -85,B 0,C 180,E1 -14643.658,E2 -14643.658} C_VEL
LIN {X 0,Y 332.23,Z 373.325,A -85,B 0,C 180,E1 -14645.452,E2 -14645.452} C_VEL
LIN {X 0,Y 331.919,Z 374.721,A -85,B 0,C 180,E1 -14647.596,E2 -14647.596} C_VEL
LIN {X 0,Y 331.893,Z 374.984,A -85,B 0,C 180,E1 -14648.901,E2 -14648.901} C_VEL
LIN {X 0,Y 331.811,Z 374.778,A -85,B 0,C 180,E1 -14650.191,E2 -14650.191} C_VEL
LIN {X 0,Y 331.89,Z 373.432,A -85,B 0,C 180,E1 -14652.343,E2 -14652.343} C_VEL
LIN {X 0,Y 332.146,Z 370.568,A -85,B 0,C 180,E1 -14654.663,E2 -14654.663} C_VEL
LIN {X 0,Y 332.504,Z 367.038,A -85,B 0,C 180,E1 -14656.556,E2 -14656.556} C_VEL
LIN {X 0,Y 332.88,Z 362.389,A -85,B 0,C 180,E1 -14658.43,E2 -14658.43} C_VEL
LIN {X 0,Y 333.555,Z 355.304,A -85,B 0,C 180,E1 -14660.602,E2 -14660.602} C_VEL
LIN {X 0,Y 334.374,Z 347.593,A -85,B 0,C 180,E1 -14662.458,E2 -14662.458} C_VEL
LIN {X 0,Y 335.268,Z 339.744,A -85,B 0,C 180,E1 -14663.984,E2 -14663.984} C_VEL
LIN {X 0,Y 336.288,Z 330.112,A -85,B 0,C 180,E1 -14665.505,E2 -14665.505} C_VEL
LIN {X 0,Y 337.378,Z 319.747,A -85,B 0,C 180,E1 -14666.823,E2 -14666.823} C_VEL
LIN {X 0,Y 338.286,Z 309.065,A -85,B 0,C 180,E1 -14667.917,E2 -14667.917} C_VEL
LIN {X 0,Y 339.114,Z 296.875,A -85,B 0,C 180,E1 -14668.887,E2 -14668.887} C_VEL
LIN {X 0,Y 339.84,Z 283.288,A -85,B 0,C 180,E1 -14669.667,E2 -14669.667} C_VEL
LIN {X 0,Y 340.399,Z 270.493,A -85,B 0,C 180,E1 -14670.148,E2 -14670.148} C_VEL
LIN {X 0,Y 341.904,Z 190.93,A -85,B 0,C 180,E1 -14671.855,E2 -14671.855} C_VEL
LIN {X 0,Y 338.972,Z 175.542,A -85,B 0,C 180,E1 -14672.362,E2 -14672.362} C_VEL
LIN {X 0,Y 335.296,Z 163.91,A -85,B 0,C 180,E1 -14672.844,E2 -14672.844} C_VEL
LIN {X 0,Y 333.778,Z 156.906,A -85,B 0,C 180,E1 -14674.907,E2 -14674.907} C_VEL
LIN {X 0,Y 333.952,Z 156.885,A -85,B 0,C 180,E1 -14677.254,E2 -14677.254} C_VEL
LIN {X 0,Y 333.805,Z 156.902,A -85,B 0,C 180,E1 -14680.923,E2 -14680.923} C_VEL
LIN {X 0,Y 333.729,Z 156.911,A -85,B 0,C 180,E1 -14684.638,E2 -14684.638} C_VEL
LIN {X 0,Y 333.686,Z 156.917,A -85,B 0,C 180,E1 -14688.601,E2 -14688.601} C_VEL
LIN {X 0,Y 333.644,Z 156.922,A -85,B 0,C 180,E1 -14692.282,E2 -14692.282} C_VEL
LIN {X 0,Y 333.65,Z 156.921,A -85,B 0,C 180,E1 -14695.096,E2 -14695.096} C_VEL
LIN {X 0,Y 332.923,Z 157.01,A -85,B 0,C 180,E1 -14696.103,E2 -14696.103} C_VEL
LIN {X 0,Y 330.032,Z 157.373,A -85,B 0,C 180,E1 -14697.742,E2 -14697.742} C_VEL
LIN {X 0,Y 327.641,Z 157.671,A -85,B 0,C 180,E1 -14699.069,E2 -14699.069} C_VEL
LIN {X 0,Y 326.656,Z 157.793,A -85,B 0,C 180,E1 -14700.097,E2 -14700.097} C_VEL
LIN {X 0,Y 326.596,Z 157.8,A -85,B 0,C 180,E1 -14700.445,E2 -14700.445} C_VEL
LIN {X 0,Y 326.604,Z 157.799,A -85,B 0,C 180,E1 -14704.02,E2 -14704.02} C_VEL
LIN {X 0,Y 326.619,Z 157.801,A -85,B 0,C 180,E1 -14707.238,E2 -14707.238} C_VEL
LIN {X 0,Y 326.541,Z 157.812,A -85,B 0,C 180,E1 -14711.125,E2 -14711.125} C_VEL
LIN {X 0,Y 326.557,Z 157.805,A -85,B 0,C 180,E1 -14713.527,E2 -14713.527} C_VEL
LIN {X 0,Y 326.57,Z 157.805,A -85,B 0,C 180,E1 -14717.03,E2 -14717.03} C_VEL
LIN {X 0,Y 326.581,Z 157.802,A -85,B 0,C 180,E1 -14721.386,E2 -14721.386} C_VEL
LIN {X 0,Y 326.618,Z 157.801,A -85,B 0,C 180,E1 -14724.853,E2 -14724.853} C_VEL
LIN {X 0,Y 326.608,Z 157.797,A -85,B 0,C 180,E1 -14727.456,E2 -14727.456} C_VEL
LIN {X 0,Y 326.58,Z 157.802,A -85,B 0,C 180,E1 -14730.334,E2 -14730.334} C_VEL
LIN {X 0,Y 326.595,Z 157.799,A -85,B 0,C 180,E1 -14733.135,E2 -14733.135} C_VEL
LIN {X 0,Y 326.592,Z 157.8,A -85,B 0,C 180,E1 -14737.211,E2 -14737.211} C_VEL
LIN {X 0,Y 326.628,Z 157.795,A -85,B 0,C 180,E1 -14741.218,E2 -14741.218} C_VEL
LIN {X 0,Y 326.717,Z 157.785,A -85,B 0,C 180,E1 -14745.467,E2 -14745.467} C_VEL
LIN {X 0,Y 326.752,Z 157.78,A -85,B 0,C 180,E1 -14748.839,E2 -14748.839} C_VEL
LIN {X 0,Y 326.921,Z 157.76,A -85,B 0,C 180,E1 -14752.59,E2 -14752.59} C_VEL
LIN {X 0,Y 326.747,Z 157.781,A -85,B 0,C 180,E1 -14755.065,E2 -14755.065} C_VEL
LIN {X 0,Y 327.005,Z 157.751,A -85,B 0,C 180,E1 -14757.537,E2 -14757.537} C_VEL
LIN {X 0,Y 327.032,Z 157.746,A -85,B 0,C 180,E1 -14761.232,E2 -14761.232} C_VEL
LIN {X 0,Y 326.752,Z 157.786,A -85,B 0,C 180,E1 -14763.7,E2 -14763.7} C_VEL
LIN {X 0,Y 326.944,Z 157.758,A -85,B 0,C 180,E1 -14766.171,E2 -14766.171} C_VEL
LIN {X 0,Y 326.787,Z 157.779,A -85,B 0,C 180,E1 -14769.908,E2 -14769.908} C_VEL
LIN {X 0,Y 326.748,Z 157.784,A -85,B 0,C 180,E1 -14773.687,E2 -14773.687} C_VEL
LIN {X 0,Y 326.637,Z 157.799,A -85,B 0,C 180,E1 -14777.532,E2 -14777.532} C_VEL
LIN {X 0,Y 326.609,Z 157.798,A -85,B 0,C 180,E1 -14780.139,E2 -14780.139} C_VEL
LIN {X 0,Y 326.633,Z 157.795,A -85,B 0,C 180,E1 -14784.131,E2 -14784.131} C_VEL
LIN {X 0,Y 326.603,Z 157.799,A -85,B 0,C 180,E1 -14788.083,E2 -14788.083} C_VEL
LIN {X 0,Y 326.576,Z 157.808,A -85,B 0,C 180,E1 -14791.098,E2 -14791.098} C_VEL
LIN {X 0,Y 326.611,Z 157.798,A -85,B 0,C 180,E1 -14794.02,E2 -14794.02} C_VEL
LIN {X 0,Y 326.627,Z 157.799,A -85,B 0,C 180,E1 -14797.237,E2 -14797.237} C_VEL
LIN {X 0,Y 326.548,Z 157.809,A -85,B 0,C 180,E1 -14801.124,E2 -14801.124} C_VEL
LIN {X 0,Y 326.564,Z 157.805,A -85,B 0,C 180,E1 -14803.526,E2 -14803.526} C_VEL
LIN {X 0,Y 326.576,Z 157.805,A -85,B 0,C 180,E1 -14807.029,E2 -14807.029} C_VEL
LIN {X 0,Y 326.586,Z 157.801,A -85,B 0,C 180,E1 -14811.386,E2 -14811.386} C_VEL
LIN {X 0,Y 326.623,Z 157.799,A -85,B 0,C 180,E1 -14814.851,E2 -14814.851} C_VEL
LIN {X 0,Y 326.612,Z 157.799,A -85,B 0,C 180,E1 -14817.455,E2 -14817.455} C_VEL
LIN {X 0,Y 326.642,Z 157.889,A -85,B 0,C 180,E1 -14819.389,E2 -14819.389} C_VEL
LIN {X 0,Y 328.815,Z 168.505,A -85,B 0,C 180,E1 -14822.297,E2 -14822.297} C_VEL
LIN {X 0,Y 330.289,Z 176.735,A -85,B 0,C 180,E1 -14824.476,E2 -14824.476} C_VEL
LIN {X 0,Y 329.264,Z 186.322,A -85,B 0,C 180,E1 -14826.819,E2 -14826.819} C_VEL
LIN {X 0,Y 334.696,Z 225.282,A -85,B 0,C 180,E1 -14828.017,E2 -14828.017} C_VEL
LIN {X 0,Y 333.288,Z 295.205,A -85,B 0,C 180,E1 -14829.558,E2 -14829.558} C_VEL
LIN {X 0,Y 332.583,Z 309.063,A -85,B 0,C 180,E1 -14830.118,E2 -14830.118} C_VEL
LIN {X 0,Y 331.599,Z 322.023,A -85,B 0,C 180,E1 -14830.902,E2 -14830.902} C_VEL
LIN {X 0,Y 330.551,Z 333.847,A -85,B 0,C 180,E1 -14831.883,E2 -14831.883} C_VEL
LIN {X 0,Y 329.367,Z 345.248,A -85,B 0,C 180,E1 -14833.098,E2 -14833.098} C_VEL
LIN {X 0,Y 328.399,Z 354.819,A -85,B 0,C 180,E1 -14834.375,E2 -14834.375} C_VEL
LIN {X 0,Y 327.564,Z 363.082,A -85,B 0,C 180,E1 -14835.715,E2 -14835.715} C_VEL
LIN {X 0,Y 326.679,Z 370.994,A -85,B 0,C 180,E1 -14837.26,E2 -14837.26} C_VEL
LIN {X 0,Y 325.86,Z 378.702,A -85,B 0,C 180,E1 -14839.122,E2 -14839.122} C_VEL
LIN {X 0,Y 325.431,Z 383.977,A -85,B 0,C 180,E1 -14840.678,E2 -14840.678} C_VEL
LIN {X 0,Y 325.106,Z 389.071,A -85,B 0,C 180,E1 -14842.547,E2 -14842.547} C_VEL
LIN {X 0,Y 324.956,Z 392.615,A -85,B 0,C 180,E1 -14844.197,E2 -14844.197} C_VEL
LIN {X 0,Y 324.938,Z 395.886,A -85,B 0,C 180,E1 -14846.279,E2 -14846.279} C_VEL
LIN {X 0,Y 324.903,Z 398.188,A -85,B 0,C 180,E1 -14848.76,E2 -14848.76} C_VEL
LIN {X 0,Y 324.95,Z 398.747,A -85,B 0,C 180,E1 -14850,E2 -14850} C_VEL
LIN {X 0,Y 324.872,Z 398.876,A -85,B 0,C 180,E1 -14851.239,E2 -14851.239} C_VEL
LIN {X 0,Y 324.894,Z 397.926,A -85,B 0,C 180,E1 -14853.721,E2 -14853.721} C_VEL
LIN {X 0,Y 324.909,Z 396,A -85,B 0,C 180,E1 -14855.721,E2 -14855.721} C_VEL
LIN {X 0,Y 325.244,Z 392.368,A -85,B 0,C 180,E1 -14858.074,E2 -14858.074} C_VEL
LIN {X 0,Y 325.781,Z 388.311,A -85,B 0,C 180,E1 -14859.938,E2 -14859.938} C_VEL
LIN {X 0,Y 326.652,Z 382.119,A -85,B 0,C 180,E1 -14862.109,E2 -14862.109} C_VEL
LIN {X 0,Y 327.917,Z 375.405,A -85,B 0,C 180,E1 -14863.952,E2 -14863.952} C_VEL
LIN {X 0,Y 329.299,Z 367.112,A -85,B 0,C 180,E1 -14865.79,E2 -14865.79} C_VEL
LIN {X 0,Y 330.684,Z 358.627,A -85,B 0,C 180,E1 -14867.31,E2 -14867.31} C_VEL
LIN {X 0,Y 332.45,Z 348.18,A -85,B 0,C 180,E1 -14868.807,E2 -14868.807} C_VEL
LIN {X 0,Y 334.272,Z 336.456,A -85,B 0,C 180,E1 -14870.138,E2 -14870.138} C_VEL
LIN {X 0,Y 335.79,Z 324.722,A -85,B 0,C 180,E1 -14871.164,E2 -14871.164} C_VEL
LIN {X 0,Y 337.098,Z 312.586,A -85,B 0,C 180,E1 -14871.961,E2 -14871.961} C_VEL
LIN {X 0,Y 338.249,Z 299.351,A -85,B 0,C 180,E1 -14872.565,E2 -14872.565} C_VEL
LIN {X 0,Y 338.843,Z 284.701,A -85,B 0,C 180,E1 -14872.966,E2 -14872.966} C_VEL
LIN {X 0,Y 340.153,Z 226.079,A -85,B 0,C 180,E1 -14874.261,E2 -14874.261} C_VEL
LIN {X 0,Y 336.788,Z 205.858,A -85,B 0,C 180,E1 -14875.068,E2 -14875.068} C_VEL
LIN {X 0,Y 332.29,Z 185.202,A -85,B 0,C 180,E1 -14876.049,E2 -14876.049} C_VEL
LIN {X 0,Y 331.954,Z 180.935,A -85,B 0,C 180,E1 -14877.225,E2 -14877.225} C_VEL
LIN {X 0,Y 329.703,Z 170.215,A -85,B 0,C 180,E1 -14880.415,E2 -14880.415} C_VEL
LIN {X 0,Y 327.545,Z 161.418,A -85,B 0,C 180,E1 -14883.194,E2 -14883.194} C_VEL
LIN {X 0,Y 326.622,Z 157.793,A -85,B 0,C 180,E1 -14884.39,E2 -14884.39} C_VEL
LIN {X 0,Y 326.625,Z 157.791,A -85,B 0,C 180,E1 -14887.237,E2 -14887.237} C_VEL
LIN {X 0,Y 326.545,Z 157.798,A -85,B 0,C 180,E1 -14891.124,E2 -14891.124} C_VEL
LIN {X 0,Y 326.561,Z 157.807,A -85,B 0,C 180,E1 -14893.526,E2 -14893.526} C_VEL
LIN {X 0,Y 326.574,Z 157.804,A -85,B 0,C 180,E1 -14897.029,E2 -14897.029} C_VEL
LIN {X 0,Y 326.583,Z 157.801,A -85,B 0,C 180,E1 -14901.385,E2 -14901.385} C_VEL
LIN {X 0,Y 326.62,Z 157.795,A -85,B 0,C 180,E1 -14904.852,E2 -14904.852} C_VEL
LIN {X 0,Y 326.61,Z 157.799,A -85,B 0,C 180,E1 -14907.455,E2 -14907.455} C_VEL
LIN {X 0,Y 326.616,Z 157.795,A -85,B 0,C 180,E1 -14910.336,E2 -14910.336} C_VEL
LIN {X 0,Y 326.602,Z 157.798,A -85,B 0,C 180,E1 -14914.508,E2 -14914.508} C_VEL
LIN {X 0,Y 326.605,Z 157.795,A -85,B 0,C 180,E1 -14918.542,E2 -14918.542} C_VEL
LIN {X 0,Y 326.629,Z 157.789,A -85,B 0,C 180,E1 -14922.468,E2 -14922.468} C_VEL
LIN {X 0,Y 326.744,Z 157.773,A -85,B 0,C 180,E1 -14926.313,E2 -14926.313} C_VEL
LIN {X 0,Y 326.784,Z 157.777,A -85,B 0,C 180,E1 -14930.092,E2 -14930.092} C_VEL
LIN {X 0,Y 326.945,Z 157.758,A -85,B 0,C 180,E1 -14933.829,E2 -14933.829} C_VEL
LIN {X 0,Y 327.011,Z 157.74,A -85,B 0,C 180,E1 -14937.536,E2 -14937.536} C_VEL
LIN {X 0,Y 327.034,Z 157.737,A -85,B 0,C 180,E1 -14941.231,E2 -14941.231} C_VEL
LIN {X 0,Y 327.043,Z 157.742,A -85,B 0,C 180,E1 -14942.463,E2 -14942.463} C_VEL
LIN {X 0,Y 326.924,Z 157.751,A -85,B 0,C 180,E1 -14946.481,E2 -14946.481} C_VEL
LIN {X 0,Y 326.784,Z 157.77,A -85,B 0,C 180,E1 -14949.906,E2 -14949.906} C_VEL
LIN {X 0,Y 326.76,Z 157.777,A -85,B 0,C 180,E1 -14953.685,E2 -14953.685} C_VEL
LIN {X 0,Y 326.665,Z 157.79,A -85,B 0,C 180,E1 -14957.529,E2 -14957.529} C_VEL
LIN {X 0,Y 326.65,Z 157.796,A -85,B 0,C 180,E1 -14960.135,E2 -14960.135} C_VEL
LIN {X 0,Y 326.649,Z 157.798,A -85,B 0,C 180,E1 -14964.128,E2 -14964.128} C_VEL
LIN {X 0,Y 326.684,Z 157.795,A -85,B 0,C 180,E1 -14966.857,E2 -14966.857} C_VEL
LIN {X 0,Y 326.638,Z 157.796,A -85,B 0,C 180,E1 -14970.61,E2 -14970.61} C_VEL
LIN {X 0,Y 326.606,Z 157.803,A -85,B 0,C 180,E1 -14974.019,E2 -14974.019} C_VEL
LIN {X 0,Y 326.626,Z 157.805,A -85,B 0,C 180,E1 -14977.238,E2 -14977.238} C_VEL
LIN {X 0,Y 326.607,Z 157.905,A -85,B 0,C 180,E1 -14981.137,E2 -14981.137} C_VEL
LIN {X 0,Y 328.432,Z 165.148,A -85,B 0,C 180,E1 -14983.608,E2 -14983.608} C_VEL
LIN {X 0,Y 336.917,Z 183.153,A -85,B 0,C 180,E1 -14984.937,E2 -14984.937} C_VEL
LIN {X 0,Y 340.404,Z 191.868,A -85,B 0,C 180,E1 -14985.485,E2 -14985.485} C_VEL
LIN {X 0,Y 341.095,Z 195.233,A -85,B 0,C 180,E1 -14985.631,E2 -14985.631} C_VEL
LIN {X 0,Y 338.968,Z 272.324,A -85,B 0,C 180,E1 -14987.334,E2 -14987.334} C_VEL
LIN {X 0,Y 338.177,Z 285.66,A -85,B 0,C 180,E1 -14987.866,E2 -14987.866} C_VEL
LIN {X 0,Y 337.203,Z 298.202,A -85,B 0,C 180,E1 -14988.616,E2 -14988.616} C_VEL
LIN {X 0,Y 335.903,Z 309.926,A -85,B 0,C 180,E1 -14989.563,E2 -14989.563} C_VEL
LIN {X 0,Y 334.394,Z 321.008,A -85,B 0,C 180,E1 -14990.718,E2 -14990.718} C_VEL
LIN {X 0,Y 332.864,Z 331.302,A -85,B 0,C 180,E1 -14992.069,E2 -14992.069} C_VEL
LIN {X 0,Y 331.29,Z 340.485,A -85,B 0,C 180,E1 -14993.559,E2 -14993.559} C_VEL
LIN {X 0,Y 329.805,Z 348.838,A -85,B 0,C 180,E1 -14995.248,E2 -14995.248} C_VEL
LIN {X 0,Y 328.327,Z 356.867,A -85,B 0,C 180,E1 -14997.283,E2 -14997.283} C_VEL
LIN {X 0,Y 327.166,Z 362.898,A -85,B 0,C 180,E1 -14999.232,E2 -14999.232} C_VEL
LIN {X 0,Y 326.398,Z 367.215,A -85,B 0,C 180,E1 -15001.022,E2 -15001.022} C_VEL
LIN {X 0,Y 325.684,Z 370.909,A -85,B 0,C 180,E1 -15003.053,E2 -15003.053} C_VEL
LIN {X 0,Y 325.182,Z 373.521,A -85,B 0,C 180,E1 -15005.191,E2 -15005.191} C_VEL
LIN {X 0,Y 324.883,Z 374.846,A -85,B 0,C 180,E1 -15007.084,E2 -15007.084} C_VEL
LIN {X 0,Y 324.806,Z 375.214,A -85,B 0,C 180,E1 -15008.497,E2 -15008.497} C_VEL
LIN {X 0,Y 324.75,Z 375.141,A -85,B 0,C 180,E1 -15009.741,E2 -15009.741} C_VEL
LIN {X 0,Y 324.725,Z 374.624,A -85,B 0,C 180,E1 -15011.056,E2 -15011.056} C_VEL
LIN {X 0,Y 324.812,Z 373.64,A -85,B 0,C 180,E1 -15012.367,E2 -15012.367} C_VEL
LIN {X 0,Y 324.909,Z 372.241,A -85,B 0,C 180,E1 -15013.668,E2 -15013.668} C_VEL
LIN {X 0,Y 325.25,Z 369.261,A -85,B 0,C 180,E1 -15015.612,E2 -15015.612} C_VEL
LIN {X 0,Y 325.593,Z 365.208,A -85,B 0,C 180,E1 -15017.535,E2 -15017.535} C_VEL
LIN {X 0,Y 326.16,Z 358.944,A -85,B 0,C 180,E1 -15019.76,E2 -15019.76} C_VEL
LIN {X 0,Y 326.949,Z 351.793,A -85,B 0,C 180,E1 -15021.726,E2 -15021.726} C_VEL
LIN {X 0,Y 327.883,Z 343.523,A -85,B 0,C 180,E1 -15023.539,E2 -15023.539} C_VEL
LIN {X 0,Y 328.854,Z 334.693,A -85,B 0,C 180,E1 -15025.096,E2 -15025.096} C_VEL
LIN {X 0,Y 330.079,Z 323.775,A -85,B 0,C 180,E1 -15026.644,E2 -15026.644} C_VEL
LIN {X 0,Y 331.118,Z 312.889,A -85,B 0,C 180,E1 -15027.872,E2 -15027.872} C_VEL
LIN {X 0,Y 332.023,Z 300.71,A -85,B 0,C 180,E1 -15028.939,E2 -15028.939} C_VEL
LIN {X 0,Y 332.848,Z 287.939,A -85,B 0,C 180,E1 -15029.773,E2 -15029.773} C_VEL
LIN {X 0,Y 333.422,Z 275.309,A -85,B 0,C 180,E1 -15030.34,E2 -15030.34} C_VEL
LIN {X 0,Y 333.858,Z 257.72,A -85,B 0,C 180,E1 -15030.792,E2 -15030.792} C_VEL
LIN {X 0,Y 335.116,Z 191.537,A -85,B 0,C 180,E1 -15032.221,E2 -15032.221} C_VEL
LIN {X 0,Y 332.386,Z 177.466,A -85,B 0,C 180,E1 -15032.699,E2 -15032.699} C_VEL
LIN {X 0,Y 328.077,Z 164.182,A -85,B 0,C 180,E1 -15033.263,E2 -15033.263} C_VEL
LIN {X 0,Y 326.774,Z 157.781,A -85,B 0,C 180,E1 -15035.206,E2 -15035.206} C_VEL
LIN {X 0,Y 326.909,Z 157.764,A -85,B 0,C 180,E1 -15037.412,E2 -15037.412} C_VEL
LIN {X 0,Y 326.745,Z 157.782,A -85,B 0,C 180,E1 -15041.162,E2 -15041.162} C_VEL
LIN {X 0,Y 326.658,Z 157.793,A -85,B 0,C 180,E1 -15044.962,E2 -15044.962} C_VEL
LIN {X 0,Y 326.633,Z 157.796,A -85,B 0,C 180,E1 -15048.83,E2 -15048.83} C_VEL
LIN {X 0,Y 326.585,Z 157.8,A -85,B 0,C 180,E1 -15052.79,E2 -15052.79} C_VEL
LIN {X 0,Y 326.591,Z 157.798,A -85,B 0,C 180,E1 -15056.866,E2 -15056.866} C_VEL
LIN {X 0,Y 326.596,Z 157.8,A -85,B 0,C 180,E1 -15060.445,E2 -15060.445} C_VEL
LIN {X 0,Y 325.984,Z 157.88,A -85,B 0,C 180,E1 -15061.473,E2 -15061.473} C_VEL
LIN {X 0,Y 323.154,Z 158.233,A -85,B 0,C 180,E1 -15063.147,E2 -15063.147} C_VEL
LIN {X 0,Y 320.713,Z 158.535,A -85,B 0,C 180,E1 -15064.503,E2 -15064.503} C_VEL
LIN {X 0,Y 319.65,Z 158.665,A -85,B 0,C 180,E1 -15065.553,E2 -15065.553} C_VEL
LIN {X 0,Y 319.557,Z 158.674,A -85,B 0,C 180,E1 -15065.909,E2 -15065.909} C_VEL
LIN {X 0,Y 319.526,Z 158.682,A -85,B 0,C 180,E1 -15069.663,E2 -15069.663} C_VEL
LIN {X 0,Y 319.517,Z 158.682,A -85,B 0,C 180,E1 -15073.461,E2 -15073.461} C_VEL
LIN {X 0,Y 319.549,Z 158.679,A -85,B 0,C 180,E1 -15077.017,E2 -15077.017} C_VEL
LIN {X 0,Y 319.544,Z 158.679,A -85,B 0,C 180,E1 -15080.371,E2 -15080.371} C_VEL
LIN {X 0,Y 319.578,Z 158.677,A -85,B 0,C 180,E1 -15084.459,E2 -15084.459} C_VEL
LIN {X 0,Y 319.524,Z 158.68,A -85,B 0,C 180,E1 -15088.138,E2 -15088.138} C_VEL
LIN {X 0,Y 319.544,Z 158.673,A -85,B 0,C 180,E1 -15091.614,E2 -15091.614} C_VEL
LIN {X 0,Y 319.526,Z 158.68,A -85,B 0,C 180,E1 -15095.298,E2 -15095.298} C_VEL
LIN {X 0,Y 319.561,Z 158.679,A -85,B 0,C 180,E1 -15098.046,E2 -15098.046} C_VEL
LIN {X 0,Y 319.575,Z 158.677,A -85,B 0,C 180,E1 -15102.069,E2 -15102.069} C_VEL
LIN {X 0,Y 319.696,Z 158.663,A -85,B 0,C 180,E1 -15106.007,E2 -15106.007} C_VEL
LIN {X 0,Y 319.735,Z 158.658,A -85,B 0,C 180,E1 -15109.873,E2 -15109.873} C_VEL
LIN {X 0,Y 319.904,Z 158.636,A -85,B 0,C 180,E1 -15113.694,E2 -15113.694} C_VEL
LIN {X 0,Y 319.951,Z 158.629,A -85,B 0,C 180,E1 -15117.483,E2 -15117.483} C_VEL
LIN {X 0,Y 320.002,Z 158.622,A -85,B 0,C 180,E1 -15121.259,E2 -15121.259} C_VEL
LIN {X 0,Y 319.702,Z 158.664,A -85,B 0,C 180,E1 -15123.782,E2 -15123.782} C_VEL
LIN {X 0,Y 319.901,Z 158.634,A -85,B 0,C 180,E1 -15126.307,E2 -15126.307} C_VEL
LIN {X 0,Y 319.74,Z 158.655,A -85,B 0,C 180,E1 -15130.128,E2 -15130.128} C_VEL
LIN {X 0,Y 319.714,Z 158.658,A -85,B 0,C 180,E1 -15133.994,E2 -15133.994} C_VEL
LIN {X 0,Y 319.591,Z 158.673,A -85,B 0,C 180,E1 -15137.931,E2 -15137.931} C_VEL
LIN {X 0,Y 319.567,Z 158.676,A -85,B 0,C 180,E1 -15141.955,E2 -15141.955} C_VEL
LIN {X 0,Y 319.572,Z 158.675,A -85,B 0,C 180,E1 -15146.094,E2 -15146.094} C_VEL
LIN {X 0,Y 319.545,Z 158.682,A -85,B 0,C 180,E1 -15148.939,E2 -15148.939} C_VEL
LIN {X 0,Y 319.527,Z 158.681,A -85,B 0,C 180,E1 -15151.863,E2 -15151.863} C_VEL
LIN {X 0,Y 319.583,Z 158.675,A -85,B 0,C 180,E1 -15155.543,E2 -15155.543} C_VEL
LIN {X 0,Y 319.532,Z 158.68,A -85,B 0,C 180,E1 -15159.662,E2 -15159.662} C_VEL
LIN {X 0,Y 319.523,Z 158.682,A -85,B 0,C 180,E1 -15163.46,E2 -15163.46} C_VEL
LIN {X 0,Y 319.555,Z 158.68,A -85,B 0,C 180,E1 -15167.016,E2 -15167.016} C_VEL
LIN {X 0,Y 319.549,Z 158.682,A -85,B 0,C 180,E1 -15170.371,E2 -15170.371} C_VEL
LIN {X 0,Y 319.584,Z 158.679,A -85,B 0,C 180,E1 -15174.457,E2 -15174.457} C_VEL
LIN {X 0,Y 319.536,Z 158.684,A -85,B 0,C 180,E1 -15178.138,E2 -15178.138} C_VEL
LIN {X 0,Y 319.57,Z 158.701,A -85,B 0,C 180,E1 -15179.059,E2 -15179.059} C_VEL
LIN {X 0,Y 321.983,Z 170.501,A -85,B 0,C 180,E1 -15182.365,E2 -15182.365} C_VEL
LIN {X 0,Y 323.277,Z 178.713,A -85,B 0,C 180,E1 -15184.572,E2 -15184.572} C_VEL
LIN {X 0,Y 322.432,Z 186.024,A -85,B 0,C 180,E1 -15186.394,E2 -15186.394} C_VEL
LIN {X 0,Y 327.922,Z 226.697,A -85,B 0,C 180,E1 -15187.677,E2 -15187.677} C_VEL
LIN {X 0,Y 326.498,Z 294.514,A -85,B 0,C 180,E1 -15189.196,E2 -15189.196} C_VEL
LIN {X 0,Y 325.821,Z 307.76,A -85,B 0,C 180,E1 -15189.728,E2 -15189.728} C_VEL
LIN {X 0,Y 324.866,Z 320.514,A -85,B 0,C 180,E1 -15190.49,E2 -15190.49} C_VEL
LIN {X 0,Y 323.797,Z 332.667,A -85,B 0,C 180,E1 -15191.492,E2 -15191.492} C_VEL
LIN {X 0,Y 322.476,Z 344.231,A -85,B 0,C 180,E1 -15192.726,E2 -15192.726} C_VEL
LIN {X 0,Y 321.385,Z 355.061,A -85,B 0,C 180,E1 -15194.195,E2 -15194.195} C_VEL
LIN {X 0,Y 320.42,Z 364.044,A -85,B 0,C 180,E1 -15195.714,E2 -15195.714} C_VEL
LIN {X 0,Y 319.394,Z 373.112,A -85,B 0,C 180,E1 -15197.611,E2 -15197.611} C_VEL
LIN {X 0,Y 318.663,Z 380.397,A -85,B 0,C 180,E1 -15199.516,E2 -15199.516} C_VEL
LIN {X 0,Y 318.237,Z 385.302,A -85,B 0,C 180,E1 -15201.107,E2 -15201.107} C_VEL
LIN {X 0,Y 317.98,Z 390.059,A -85,B 0,C 180,E1 -15203.018,E2 -15203.018} C_VEL
LIN {X 0,Y 317.832,Z 393.673,A -85,B 0,C 180,E1 -15204.925,E2 -15204.925} C_VEL
LIN {X 0,Y 317.844,Z 395.525,A -85,B 0,C 180,E1 -15206.196,E2 -15206.196} C_VEL
LIN {X 0,Y 317.797,Z 396.9,A -85,B 0,C 180,E1 -15207.465,E2 -15207.465} C_VEL
LIN {X 0,Y 317.81,Z 397.873,A -85,B 0,C 180,E1 -15208.733,E2 -15208.733} C_VEL
LIN {X 0,Y 317.855,Z 398.454,A -85,B 0,C 180,E1 -15210,E2 -15210} C_VEL
LIN {X 0,Y 317.781,Z 398.624,A -85,B 0,C 180,E1 -15211.267,E2 -15211.267} C_VEL
LIN {X 0,Y 317.777,Z 398.364,A -85,B 0,C 180,E1 -15212.535,E2 -15212.535} C_VEL
LIN {X 0,Y 317.801,Z 397.719,A -85,B 0,C 180,E1 -15213.804,E2 -15213.804} C_VEL
LIN {X 0,Y 317.889,Z 395.25,A -85,B 0,C 180,E1 -15216.346,E2 -15216.346} C_VEL
LIN {X 0,Y 318.199,Z 392.274,A -85,B 0,C 180,E1 -15218.254,E2 -15218.254} C_VEL
LIN {X 0,Y 318.764,Z 388.276,A -85,B 0,C 180,E1 -15220.159,E2 -15220.159} C_VEL
LIN {X 0,Y 319.7,Z 382.169,A -85,B 0,C 180,E1 -15222.376,E2 -15222.376} C_VEL
LIN {X 0,Y 321.021,Z 375.523,A -85,B 0,C 180,E1 -15224.258,E2 -15224.258} C_VEL
LIN {X 0,Y 322.263,Z 368.791,A -85,B 0,C 180,E1 -15225.819,E2 -15225.819} C_VEL
LIN {X 0,Y 323.608,Z 360.715,A -85,B 0,C 180,E1 -15227.374,E2 -15227.374} C_VEL
LIN {X 0,Y 325.387,Z 350.882,A -85,B 0,C 180,E1 -15228.904,E2 -15228.904} C_VEL
LIN {X 0,Y 327.205,Z 339.901,A -85,B 0,C 180,E1 -15230.264,E2 -15230.264} C_VEL
LIN {X 0,Y 328.978,Z 327.434,A -85,B 0,C 180,E1 -15231.459,E2 -15231.459} C_VEL
LIN {X 0,Y 330.483,Z 315.17,A -85,B 0,C 180,E1 -15232.341,E2 -15232.341} C_VEL
LIN {X 0,Y 331.663,Z 302.226,A -85,B 0,C 180,E1 -15232.998,E2 -15232.998} C_VEL
LIN {X 0,Y 332.416,Z 290.001,A -85,B 0,C 180,E1 -15233.395,E2 -15233.395} C_VEL
LIN {X 0,Y 333.926,Z 227.21,A -85,B 0,C 180,E1 -15234.813,E2 -15234.813} C_VEL
LIN {X 0,Y 330.778,Z 208.055,A -85,B 0,C 180,E1 -15235.597,E2 -15235.597} C_VEL
LIN {X 0,Y 326.326,Z 187.641,A -85,B 0,C 180,E1 -15236.585,E2 -15236.585} C_VEL
LIN {X 0,Y 325.488,Z 184.851,A -85,B 0,C 180,E1 -15236.786,E2 -15236.786} C_VEL
LIN {X 0,Y 323.401,Z 174.188,A -85,B 0,C 180,E1 -15239.988,E2 -15239.988} C_VEL
LIN {X 0,Y 321.315,Z 165.465,A -85,B 0,C 180,E1 -15242.775,E2 -15242.775} C_VEL
LIN {X 0,Y 319.603,Z 158.67,A -85,B 0,C 180,E1 -15245.121,E2 -15245.121} C_VEL
LIN {X 0,Y 319.534,Z 158.678,A -85,B 0,C 180,E1 -15248.013,E2 -15248.013} C_VEL
LIN {X 0,Y 319.506,Z 158.677,A -85,B 0,C 180,E1 -15251.592,E2 -15251.592} C_VEL
LIN {X 0,Y 319.488,Z 158.687,A -85,B 0,C 180,E1 -15254.743,E2 -15254.743} C_VEL
LIN {X 0,Y 319.552,Z 158.678,A -85,B 0,C 180,E1 -15257.015,E2 -15257.015} C_VEL
LIN {X 0,Y 319.547,Z 158.68,A -85,B 0,C 180,E1 -15260.37,E2 -15260.37} C_VEL
LIN {X 0,Y 319.58,Z 158.676,A -85,B 0,C 180,E1 -15264.457,E2 -15264.457} C_VEL
LIN {X 0,Y 319.526,Z 158.682,A -85,B 0,C 180,E1 -15268.137,E2 -15268.137} C_VEL
LIN {X 0,Y 319.571,Z 158.675,A -85,B 0,C 180,E1 -15271.604,E2 -15271.604} C_VEL
LIN {X 0,Y 319.541,Z 158.679,A -85,B 0,C 180,E1 -15275.298,E2 -15275.298} C_VEL
LIN {X 0,Y 319.562,Z 158.668,A -85,B 0,C 180,E1 -15278.045,E2 -15278.045} C_VEL
LIN {X 0,Y 319.585,Z 158.666,A -85,B 0,C 180,E1 -15282.068,E2 -15282.068} C_VEL
LIN {X 0,Y 319.711,Z 158.652,A -85,B 0,C 180,E1 -15286.006,E2 -15286.006} C_VEL
LIN {X 0,Y 319.736,Z 158.657,A -85,B 0,C 180,E1 -15289.872,E2 -15289.872} C_VEL
LIN {X 0,Y 319.902,Z 158.633,A -85,B 0,C 180,E1 -15293.693,E2 -15293.693} C_VEL
LIN {X 0,Y 319.957,Z 158.618,A -85,B 0,C 180,E1 -15297.481,E2 -15297.481} C_VEL
LIN {X 0,Y 320.004,Z 158.612,A -85,B 0,C 180,E1 -15301.258,E2 -15301.258} C_VEL
LIN {X 0,Y 319.73,Z 158.658,A -85,B 0,C 180,E1 -15303.78,E2 -15303.78} C_VEL
LIN {X 0,Y 319.889,Z 158.628,A -85,B 0,C 180,E1 -15306.462,E2 -15306.462} C_VEL
LIN {X 0,Y 319.737,Z 158.647,A -85,B 0,C 180,E1 -15310.127,E2 -15310.127} C_VEL
LIN {X 0,Y 319.733,Z 158.651,A -85,B 0,C 180,E1 -15313.991,E2 -15313.991} C_VEL
LIN {X 0,Y 319.625,Z 158.665,A -85,B 0,C 180,E1 -15317.928,E2 -15317.928} C_VEL
LIN {X 0,Y 319.598,Z 158.677,A -85,B 0,C 180,E1 -15320.599,E2 -15320.599} C_VEL
LIN {X 0,Y 319.603,Z 158.672,A -85,B 0,C 180,E1 -15324.695,E2 -15324.695} C_VEL
LIN {X 0,Y 319.615,Z 158.67,A -85,B 0,C 180,E1 -15328.411,E2 -15328.411} C_VEL
LIN {X 0,Y 319.531,Z 158.684,A -85,B 0,C 180,E1 -15331.861,E2 -15331.861} C_VEL
LIN {X 0,Y 319.578,Z 158.68,A -85,B 0,C 180,E1 -15335.542,E2 -15335.542} C_VEL
LIN {X 0,Y 319.571,Z 158.681,A -85,B 0,C 180,E1 -15338.007,E2 -15338.007} C_VEL
LIN {X 0,Y 319.578,Z 158.692,A -85,B 0,C 180,E1 -15340.446,E2 -15340.446} C_VEL
LIN {X 0,Y 321.293,Z 165.424,A -85,B 0,C 180,E1 -15342.824,E2 -15342.824} C_VEL
LIN {X 0,Y 329.605,Z 182.67,A -85,B 0,C 180,E1 -15344.184,E2 -15344.184} C_VEL
LIN {X 0,Y 334.411,Z 194.067,A -85,B 0,C 180,E1 -15344.963,E2 -15344.963} C_VEL
LIN {X 0,Y 334.887,Z 197.48,A -85,B 0,C 180,E1 -15345.094,E2 -15345.094} C_VEL
LIN {X 0,Y 332.653,Z 272.989,A -85,B 0,C 180,E1 -15346.792,E2 -15346.792} C_VEL
LIN {X 0,Y 331.841,Z 286.202,A -85,B 0,C 180,E1 -15347.334,E2 -15347.334} C_VEL
LIN {X 0,Y 330.87,Z 298.062,A -85,B 0,C 180,E1 -15348.055,E2 -15348.055} C_VEL
LIN {X 0,Y 329.495,Z 309.879,A -85,B 0,C 180,E1 -15349.013,E2 -15349.013} C_VEL
LIN {X 0,Y 327.918,Z 321.126,A -85,B 0,C 180,E1 -15350.201,E2 -15350.201} C_VEL
LIN {X 0,Y 326.143,Z 332.418,A -85,B 0,C 180,E1 -15351.718,E2 -15351.718} C_VEL
LIN {X 0,Y 324.493,Z 341.523,A -85,B 0,C 180,E1 -15353.259,E2 -15353.259} C_VEL
LIN {X 0,Y 322.806,Z 350.446,A -85,B 0,C 180,E1 -15355.145,E2 -15355.145} C_VEL
LIN {X 0,Y 321.287,Z 358.189,A -85,B 0,C 180,E1 -15357.221,E2 -15357.221} C_VEL
LIN {X 0,Y 320.088,Z 364.042,A -85,B 0,C 180,E1 -15359.244,E2 -15359.244} C_VEL
LIN {X 0,Y 319.299,Z 368.1,A -85,B 0,C 180,E1 -15361.038,E2 -15361.038} C_VEL
LIN {X 0,Y 318.796,Z 370.576,A -85,B 0,C 180,E1 -15362.422,E2 -15362.422} C_VEL
LIN {X 0,Y 318.415,Z 372.535,A -85,B 0,C 180,E1 -15363.805,E2 -15363.805} C_VEL
LIN {X 0,Y 318.107,Z 373.952,A -85,B 0,C 180,E1 -15365.18,E2 -15365.18} C_VEL
LIN {X 0,Y 317.852,Z 374.924,A -85,B 0,C 180,E1 -15366.547,E2 -15366.547} C_VEL
LIN {X 0,Y 317.712,Z 375.468,A -85,B 0,C 180,E1 -15368.288,E2 -15368.288} C_VEL
LIN {X 0,Y 317.647,Z 375.065,A -85,B 0,C 180,E1 -15370.617,E2 -15370.617} C_VEL
LIN {X 0,Y 317.696,Z 374.168,A -85,B 0,C 180,E1 -15372.031,E2 -15372.031} C_VEL
LIN {X 0,Y 317.78,Z 372.927,A -85,B 0,C 180,E1 -15373.291,E2 -15373.291} C_VEL
LIN {X 0,Y 318.087,Z 370.139,A -85,B 0,C 180,E1 -15375.281,E2 -15375.281} C_VEL
LIN {X 0,Y 318.445,Z 366.283,A -85,B 0,C 180,E1 -15377.25,E2 -15377.25} C_VEL
LIN {X 0,Y 318.909,Z 361.262,A -85,B 0,C 180,E1 -15379.204,E2 -15379.204} C_VEL
LIN {X 0,Y 319.629,Z 354.915,A -85,B 0,C 180,E1 -15381.146,E2 -15381.146} C_VEL
LIN {X 0,Y 320.474,Z 346.993,A -85,B 0,C 180,E1 -15383.073,E2 -15383.073} C_VEL
LIN {X 0,Y 321.446,Z 338.85,A -85,B 0,C 180,E1 -15384.669,E2 -15384.669} C_VEL
LIN {X 0,Y 322.622,Z 328.891,A -85,B 0,C 180,E1 -15386.253,E2 -15386.253} C_VEL
LIN {X 0,Y 323.657,Z 319.124,A -85,B 0,C 180,E1 -15387.511,E2 -15387.511} C_VEL
LIN {X 0,Y 324.648,Z 308.573,A -85,B 0,C 180,E1 -15388.607,E2 -15388.607} C_VEL
LIN {X 0,Y 325.524,Z 296.011,A -85,B 0,C 180,E1 -15389.614,E2 -15389.614} C_VEL
LIN {X 0,Y 326.286,Z 282.687,A -85,B 0,C 180,E1 -15390.386,E2 -15390.386} C_VEL
LIN {X 0,Y 326.806,Z 270.419,A -85,B 0,C 180,E1 -15390.847,E2 -15390.847} C_VEL
LIN {X 0,Y 328.453,Z 192.965,A -85,B 0,C 180,E1 -15392.568,E2 -15392.568} C_VEL
LIN {X 0,Y 325.961,Z 179.783,A -85,B 0,C 180,E1 -15393.023,E2 -15393.023} C_VEL
LIN {X 0,Y 321.606,Z 166.633,A -85,B 0,C 180,E1 -15393.602,E2 -15393.602} C_VEL
LIN {X 0,Y 320.817,Z 164.395,A -85,B 0,C 180,E1 -15393.719,E2 -15393.719} C_VEL
LIN {X 0,Y 319.793,Z 158.653,A -85,B 0,C 180,E1 -15395.518,E2 -15395.518} C_VEL
LIN {X 0,Y 319.816,Z 158.645,A -85,B 0,C 180,E1 -15398.849,E2 -15398.849} C_VEL
LIN {X 0,Y 319.651,Z 158.666,A -85,B 0,C 180,E1 -15402.701,E2 -15402.701} C_VEL
LIN {X 0,Y 319.61,Z 158.673,A -85,B 0,C 180,E1 -15405.3,E2 -15405.3} C_VEL
LIN {X 0,Y 319.567,Z 158.678,A -85,B 0,C 180,E1 -15409.262,E2 -15409.262} C_VEL
LIN {X 0,Y 319.526,Z 158.683,A -85,B 0,C 180,E1 -15413.323,E2 -15413.323} C_VEL
LIN {X 0,Y 319.545,Z 158.674,A -85,B 0,C 180,E1 -15416.096,E2 -15416.096} C_VEL
LIN {X 0,Y 319.521,Z 158.681,A -85,B 0,C 180,E1 -15418.941,E2 -15418.941} C_VEL
LIN {X 0,Y 319.521,Z 158.682,A -85,B 0,C 180,E1 -15421.864,E2 -15421.864} C_VEL
LIN {X 0,Y 319.575,Z 158.674,A -85,B 0,C 180,E1 -15425.543,E2 -15425.543} C_VEL
LIN {X 0,Y 319.557,Z 158.674,A -85,B 0,C 180,E1 -15425.909,E2 -15425.909} C_VEL
LIN {X 0,Y 318.861,Z 158.765,A -85,B 0,C 180,E1 -15426.961,E2 -15426.961} C_VEL
LIN {X 0,Y 315.963,Z 159.125,A -85,B 0,C 180,E1 -15428.671,E2 -15428.671} C_VEL
LIN {X 0,Y 313.528,Z 159.428,A -85,B 0,C 180,E1 -15430.058,E2 -15430.058} C_VEL
LIN {X 0,Y 312.5,Z 159.56,A -85,B 0,C 180,E1 -15431.133,E2 -15431.133} C_VEL
LIN {X 0,Y 312.424,Z 159.563,A -85,B 0,C 180,E1 -15431.497,E2 -15431.497} C_VEL
LIN {X 0,Y 312.448,Z 159.561,A -85,B 0,C 180,E1 -15434.211,E2 -15434.211} C_VEL
LIN {X 0,Y 312.452,Z 159.557,A -85,B 0,C 180,E1 -15437.926,E2 -15437.926} C_VEL
LIN {X 0,Y 312.482,Z 159.558,A -85,B 0,C 180,E1 -15441.924,E2 -15441.924} C_VEL
LIN {X 0,Y 312.53,Z 159.553,A -85,B 0,C 180,E1 -15444.221,E2 -15444.221} C_VEL
LIN {X 0,Y 312.501,Z 159.553,A -85,B 0,C 180,E1 -15447.334,E2 -15447.334} C_VEL
LIN {X 0,Y 312.484,Z 159.552,A -85,B 0,C 180,E1 -15451.3,E2 -15451.3} C_VEL
LIN {X 0,Y 312.516,Z 159.556,A -85,B 0,C 180,E1 -15454.706,E2 -15454.706} C_VEL
LIN {X 0,Y 312.54,Z 159.551,A -85,B 0,C 180,E1 -15457.526,E2 -15457.526} C_VEL
LIN {X 0,Y 312.54,Z 159.55,A -85,B 0,C 180,E1 -15461.651,E2 -15461.651} C_VEL
LIN {X 0,Y 312.639,Z 159.54,A -85,B 0,C 180,E1 -15465.684,E2 -15465.684} C_VEL
LIN {X 0,Y 312.684,Z 159.534,A -85,B 0,C 180,E1 -15469.642,E2 -15469.642} C_VEL
LIN {X 0,Y 312.803,Z 159.521,A -85,B 0,C 180,E1 -15472.253,E2 -15472.253} C_VEL
LIN {X 0,Y 312.689,Z 159.533,A -85,B 0,C 180,E1 -15474.843,E2 -15474.843} C_VEL
LIN {X 0,Y 312.97,Z 159.496,A -85,B 0,C 180,E1 -15478.714,E2 -15478.714} C_VEL
LIN {X 0,Y 312.971,Z 159.497,A -85,B 0,C 180,E1 -15481.287,E2 -15481.287} C_VEL
LIN {X 0,Y 312.688,Z 159.534,A -85,B 0,C 180,E1 -15485.159,E2 -15485.159} C_VEL
LIN {X 0,Y 312.799,Z 159.521,A -85,B 0,C 180,E1 -15487.748,E2 -15487.748} C_VEL
LIN {X 0,Y 312.666,Z 159.54,A -85,B 0,C 180,E1 -15491.672,E2 -15491.672} C_VEL
LIN {X 0,Y 312.619,Z 159.541,A -85,B 0,C 180,E1 -15494.829,E2 -15494.829} C_VEL
LIN {X 0,Y 312.548,Z 159.553,A -85,B 0,C 180,E1 -15499.191,E2 -15499.191} C_VEL
LIN {X 0,Y 312.525,Z 159.554,A -85,B 0,C 180,E1 -15502.778,E2 -15502.778} C_VEL
LIN {X 0,Y 312.532,Z 159.552,A -85,B 0,C 180,E1 -15505.907,E2 -15505.907} C_VEL
LIN {X 0,Y 312.499,Z 159.557,A -85,B 0,C 180,E1 -15509.656,E2 -15509.656} C_VEL
LIN {X 0,Y 312.524,Z 159.554,A -85,B 0,C 180,E1 -15513.689,E2 -15513.689} C_VEL
LIN {X 0,Y 312.518,Z 159.555,A -85,B 0,C 180,E1 -15517.387,E2 -15517.387} C_VEL
LIN {X 0,Y 312.445,Z 159.568,A -85,B 0,C 180,E1 -15520.717,E2 -15520.717} C_VEL
LIN {X 0,Y 312.454,Z 159.564,A -85,B 0,C 180,E1 -15524.21,E2 -15524.21} C_VEL
LIN {X 0,Y 312.458,Z 159.562,A -85,B 0,C 180,E1 -15527.925,E2 -15527.925} C_VEL
LIN {X 0,Y 312.488,Z 159.558,A -85,B 0,C 180,E1 -15531.922,E2 -15531.922} C_VEL
LIN {X 0,Y 312.535,Z 159.556,A -85,B 0,C 180,E1 -15534.22,E2 -15534.22} C_VEL
LIN {X 0,Y 312.509,Z 159.556,A -85,B 0,C 180,E1 -15537.334,E2 -15537.334} C_VEL
LIN {X 0,Y 312.529,Z 159.759,A -85,B 0,C 180,E1 -15538.784,E2 -15538.784} C_VEL
LIN {X 0,Y 314.637,Z 169.797,A -85,B 0,C 180,E1 -15541.68,E2 -15541.68} C_VEL
LIN {X 0,Y 316.291,Z 179.34,A -85,B 0,C 180,E1 -15544.323,E2 -15544.323} C_VEL
LIN {X 0,Y 315.571,Z 185.773,A -85,B 0,C 180,E1 -15545.964,E2 -15545.964} C_VEL
LIN {X 0,Y 321.145,Z 226.641,A -85,B 0,C 180,E1 -15547.293,E2 -15547.293} C_VEL
LIN {X 0,Y 319.678,Z 294.772,A -85,B 0,C 180,E1 -15548.857,E2 -15548.857} C_VEL
LIN {X 0,Y 318.915,Z 308.606,A -85,B 0,C 180,E1 -15549.438,E2 -15549.438} C_VEL
LIN {X 0,Y 317.957,Z 321.053,A -85,B 0,C 180,E1 -15550.216,E2 -15550.216} C_VEL
LIN {X 0,Y 316.856,Z 332.988,A -85,B 0,C 180,E1 -15551.239,E2 -15551.239} C_VEL
LIN {X 0,Y 315.499,Z 344.446,A -85,B 0,C 180,E1 -15552.499,E2 -15552.499} C_VEL
LIN {X 0,Y 314.407,Z 355.079,A -85,B 0,C 180,E1 -15553.986,E2 -15553.986} C_VEL
LIN {X 0,Y 313.277,Z 364.909,A -85,B 0,C 180,E1 -15555.713,E2 -15555.713} C_VEL
LIN {X 0,Y 312.253,Z 373.788,A -85,B 0,C 180,E1 -15557.653,E2 -15557.653} C_VEL
LIN {X 0,Y 311.543,Z 380.859,A -85,B 0,C 180,E1 -15559.603,E2 -15559.603} C_VEL
LIN {X 0,Y 311.084,Z 386.504,A -85,B 0,C 180,E1 -15561.555,E2 -15561.555} C_VEL
LIN {X 0,Y 310.832,Z 390.923,A -85,B 0,C 180,E1 -15563.508,E2 -15563.508} C_VEL
LIN {X 0,Y 310.746,Z 393.251,A -85,B 0,C 180,E1 -15564.809,E2 -15564.809} C_VEL
LIN {X 0,Y 310.752,Z 395.142,A -85,B 0,C 180,E1 -15566.109,E2 -15566.109} C_VEL
LIN {X 0,Y 310.718,Z 396.555,A -85,B 0,C 180,E1 -15567.407,E2 -15567.407} C_VEL
LIN {X 0,Y 310.721,Z 397.552,A -85,B 0,C 180,E1 -15568.704,E2 -15568.704} C_VEL
LIN {X 0,Y 310.761,Z 398.156,A -85,B 0,C 180,E1 -15570,E2 -15570} C_VEL
LIN {X 0,Y 310.693,Z 398.363,A -85,B 0,C 180,E1 -15571.296,E2 -15571.296} C_VEL
LIN {X 0,Y 310.699,Z 398.141,A -85,B 0,C 180,E1 -15572.593,E2 -15572.593} C_VEL
LIN {X 0,Y 310.712,Z 397.519,A -85,B 0,C 180,E1 -15573.891,E2 -15573.891} C_VEL
LIN {X 0,Y 310.819,Z 395.11,A -85,B 0,C 180,E1 -15576.491,E2 -15576.491} C_VEL
LIN {X 0,Y 311.146,Z 392.178,A -85,B 0,C 180,E1 -15578.442,E2 -15578.442} C_VEL
LIN {X 0,Y 311.737,Z 388.234,A -85,B 0,C 180,E1 -15580.39,E2 -15580.39} C_VEL
LIN {X 0,Y 312.569,Z 383.181,A -85,B 0,C 180,E1 -15582.334,E2 -15582.334} C_VEL
LIN {X 0,Y 313.888,Z 376.864,A -85,B 0,C 180,E1 -15584.258,E2 -15584.258} C_VEL
LIN {X 0,Y 315.393,Z 369.17,A -85,B 0,C 180,E1 -15586.132,E2 -15586.132} C_VEL
LIN {X 0,Y 316.443,Z 363.07,A -85,B 0,C 180,E1 -15587.38,E2 -15587.38} C_VEL
LIN {X 0,Y 318.256,Z 353.41,A -85,B 0,C 180,E1 -15589.009,E2 -15589.009} C_VEL
LIN {X 0,Y 320.16,Z 343.069,A -85,B 0,C 180,E1 -15590.394,E2 -15590.394} C_VEL
LIN {X 0,Y 321.912,Z 331.635,A -85,B 0,C 180,E1 -15591.618,E2 -15591.618} C_VEL
LIN {X 0,Y 323.556,Z 319.665,A -85,B 0,C 180,E1 -15592.594,E2 -15592.594} C_VEL
LIN {X 0,Y 325.002,Z 306.421,A -85,B 0,C 180,E1 -15593.37,E2 -15593.37} C_VEL
LIN {X 0,Y 326.051,Z 293.231,A -85,B 0,C 180,E1 -15593.88,E2 -15593.88} C_VEL
LIN {X 0,Y 327.726,Z 228.061,A -85,B 0,C 180,E1 -15595.397,E2 -15595.397} C_VEL
LIN {X 0,Y 324.652,Z 209.315,A -85,B 0,C 180,E1 -15596.2,E2 -15596.2} C_VEL
LIN {X 0,Y 320.436,Z 189.978,A -85,B 0,C 180,E1 -15597.167,E2 -15597.167} C_VEL
LIN {X 0,Y 318.32,Z 184.672,A -85,B 0,C 180,E1 -15597.551,E2 -15597.551} C_VEL
LIN {X 0,Y 316.271,Z 174.414,A -85,B 0,C 180,E1 -15600.737,E2 -15600.737} C_VEL
LIN {X 0,Y 314.072,Z 165.441,A -85,B 0,C 180,E1 -15603.73,E2 -15603.73} C_VEL
LIN {X 0,Y 312.532,Z 159.557,A -85,B 0,C 180,E1 -15605.835,E2 -15605.835} C_VEL
LIN {X 0,Y 312.496,Z 159.564,A -85,B 0,C 180,E1 -15609.029,E2 -15609.029} C_VEL
LIN {X 0,Y 312.467,Z 159.564,A -85,B 0,C 180,E1 -15612.435,E2 -15612.435} C_VEL
LIN {X 0,Y 312.458,Z 159.563,A -85,B 0,C 180,E1 -15616.035,E2 -15616.035} C_VEL
LIN {X 0,Y 312.457,Z 159.563,A -85,B 0,C 180,E1 -15619.885,E2 -15619.885} C_VEL
LIN {X 0,Y 312.535,Z 159.554,A -85,B 0,C 180,E1 -15624.051,E2 -15624.051} C_VEL
LIN {X 0,Y 312.503,Z 159.557,A -85,B 0,C 180,E1 -15627.333,E2 -15627.333} C_VEL
LIN {X 0,Y 312.506,Z 159.556,A -85,B 0,C 180,E1 -15631.292,E2 -15631.292} C_VEL
LIN {X 0,Y 312.523,Z 159.554,A -85,B 0,C 180,E1 -15634.705,E2 -15634.705} C_VEL
LIN {X 0,Y 312.54,Z 159.54,A -85,B 0,C 180,E1 -15637.525,E2 -15637.525} C_VEL
LIN {X 0,Y 312.546,Z 159.543,A -85,B 0,C 180,E1 -15641.65,E2 -15641.65} C_VEL
LIN {X 0,Y 312.653,Z 159.536,A -85,B 0,C 180,E1 -15645.684,E2 -15645.684} C_VEL
LIN {X 0,Y 312.686,Z 159.536,A -85,B 0,C 180,E1 -15649.641,E2 -15649.641} C_VEL
LIN {X 0,Y 312.798,Z 159.51,A -85,B 0,C 180,E1 -15652.252,E2 -15652.252} C_VEL
LIN {X 0,Y 312.691,Z 159.531,A -85,B 0,C 180,E1 -15654.841,E2 -15654.841} C_VEL
LIN {X 0,Y 312.98,Z 159.495,A -85,B 0,C 180,E1 -15658.713,E2 -15658.713} C_VEL
LIN {X 0,Y 312.932,Z 159.499,A -85,B 0,C 180,E1 -15662.574,E2 -15662.574} C_VEL
LIN {X 0,Y 312.844,Z 159.506,A -85,B 0,C 180,E1 -15666.449,E2 -15666.449} C_VEL
LIN {X 0,Y 312.752,Z 159.526,A -85,B 0,C 180,E1 -15669.05,E2 -15669.05} C_VEL
LIN {X 0,Y 312.636,Z 159.543,A -85,B 0,C 180,E1 -15672.99,E2 -15672.99} C_VEL
LIN {X 0,Y 312.622,Z 159.541,A -85,B 0,C 180,E1 -15675.65,E2 -15675.65} C_VEL
LIN {X 0,Y 312.565,Z 159.552,A -85,B 0,C 180,E1 -15679.71,E2 -15679.71} C_VEL
LIN {X 0,Y 312.526,Z 159.553,A -85,B 0,C 180,E1 -15682.78,E2 -15682.78} C_VEL
LIN {X 0,Y 312.582,Z 159.553,A -85,B 0,C 180,E1 -15686.722,E2 -15686.722} C_VEL
LIN {X 0,Y 312.544,Z 159.555,A -85,B 0,C 180,E1 -15689.649,E2 -15689.649} C_VEL
LIN {X 0,Y 312.518,Z 159.557,A -85,B 0,C 180,E1 -15693.688,E2 -15693.688} C_VEL
LIN {X 0,Y 312.535,Z 159.56,A -85,B 0,C 180,E1 -15697.383,E2 -15697.383} C_VEL
LIN {X 0,Y 312.543,Z 159.661,A -85,B 0,C 180,E1 -15699.766,E2 -15699.766} C_VEL
LIN {X 0,Y 314.13,Z 165.731,A -85,B 0,C 180,E1 -15701.996,E2 -15701.996} C_VEL
LIN {X 0,Y 322.976,Z 183.691,A -85,B 0,C 180,E1 -15703.497,E2 -15703.497} C_VEL
LIN {X 0,Y 328.508,Z 196.478,A -85,B 0,C 180,E1 -15704.424,E2 -15704.424} C_VEL
LIN {X 0,Y 328.697,Z 200.483,A -85,B 0,C 180,E1 -15704.546,E2 -15704.546} C_VEL
LIN {X 0,Y 326.413,Z 273.151,A -85,B 0,C 180,E1 -15706.21,E2 -15706.21} C_VEL
LIN {X 0,Y 325.561,Z 286.179,A -85,B 0,C 180,E1 -15706.749,E2 -15706.749} C_VEL
LIN {X 0,Y 324.492,Z 298.865,A -85,B 0,C 180,E1 -15707.538,E2 -15707.538} C_VEL
LIN {X 0,Y 323.136,Z 309.842,A -85,B 0,C 180,E1 -15708.444,E2 -15708.444} C_VEL
LIN {X 0,Y 321.487,Z 321.128,A -85,B 0,C 180,E1 -15709.65,E2 -15709.65} C_VEL
LIN {X 0,Y 319.815,Z 331.31,A -85,B 0,C 180,E1 -15711.021,E2 -15711.021} C_VEL
LIN {X 0,Y 318.292,Z 339.561,A -85,B 0,C 180,E1 -15712.382,E2 -15712.382} C_VEL
LIN {X 0,Y 316.684,Z 347.54,A -85,B 0,C 180,E1 -15713.978,E2 -15713.978} C_VEL
LIN {X 0,Y 315.208,Z 354.977,A -85,B 0,C 180,E1 -15715.814,E2 -15715.814} C_VEL
LIN {X 0,Y 313.988,Z 360.538,A -85,B 0,C 180,E1 -15717.507,E2 -15717.507} C_VEL
LIN {X 0,Y 312.84,Z 366.072,A -85,B 0,C 180,E1 -15719.638,E2 -15719.638} C_VEL
LIN {X 0,Y 311.919,Z 370.218,A -85,B 0,C 180,E1 -15721.76,E2 -15721.76} C_VEL
LIN {X 0,Y 311.486,Z 372.305,A -85,B 0,C 180,E1 -15723.176,E2 -15723.176} C_VEL
LIN {X 0,Y 311.118,Z 373.934,A -85,B 0,C 180,E1 -15724.631,E2 -15724.631} C_VEL
LIN {X 0,Y 310.844,Z 374.963,A -85,B 0,C 180,E1 -15725.985,E2 -15725.985} C_VEL
LIN {X 0,Y 310.638,Z 375.723,A -85,B 0,C 180,E1 -15728.062,E2 -15728.062} C_VEL
LIN {X 0,Y 310.566,Z 375.47,A -85,B 0,C 180,E1 -15730.157,E2 -15730.157} C_VEL
LIN {X 0,Y 310.588,Z 374.519,A -85,B 0,C 180,E1 -15731.872,E2 -15731.872} C_VEL
LIN {X 0,Y 310.811,Z 371.962,A -85,B 0,C 180,E1 -15734.256,E2 -15734.256} C_VEL
LIN {X 0,Y 311.171,Z 368.8,A -85,B 0,C 180,E1 -15736.208,E2 -15736.208} C_VEL
LIN {X 0,Y 311.569,Z 364.251,A -85,B 0,C 180,E1 -15738.287,E2 -15738.287} C_VEL
LIN {X 0,Y 312.176,Z 358.604,A -85,B 0,C 180,E1 -15740.279,E2 -15740.279} C_VEL
LIN {X 0,Y 313.014,Z 351.539,A -85,B 0,C 180,E1 -15742.258,E2 -15742.258} C_VEL
LIN {X 0,Y 313.881,Z 344.307,A -85,B 0,C 180,E1 -15743.895,E2 -15743.895} C_VEL
LIN {X 0,Y 315.027,Z 334.54,A -85,B 0,C 180,E1 -15745.682,E2 -15745.682} C_VEL
LIN {X 0,Y 316.208,Z 324.676,A -85,B 0,C 180,E1 -15747.134,E2 -15747.134} C_VEL
LIN {X 0,Y 317.327,Z 313.452,A -85,B 0,C 180,E1 -15748.46,E2 -15748.46} C_VEL
LIN {X 0,Y 318.366,Z 300.838,A -85,B 0,C 180,E1 -15749.605,E2 -15749.605} C_VEL
LIN {X 0,Y 319.221,Z 287.947,A -85,B 0,C 180,E1 -15750.473,E2 -15750.473} C_VEL
LIN {X 0,Y 319.855,Z 274.939,A -85,B 0,C 180,E1 -15751.063,E2 -15751.063} C_VEL
LIN {X 0,Y 320.328,Z 256.39,A -85,B 0,C 180,E1 -15751.543,E2 -15751.543} C_VEL
LIN {X 0,Y 321.69,Z 193.644,A -85,B 0,C 180,E1 -15752.952,E2 -15752.952} C_VEL
LIN {X 0,Y 319.35,Z 181.506,A -85,B 0,C 180,E1 -15753.386,E2 -15753.386} C_VEL
LIN {X 0,Y 315.189,Z 169.03,A -85,B 0,C 180,E1 -15753.952,E2 -15753.952} C_VEL
LIN {X 0,Y 313.619,Z 164.66,A -85,B 0,C 180,E1 -15754.177,E2 -15754.177} C_VEL
LIN {X 0,Y 312.798,Z 159.528,A -85,B 0,C 180,E1 -15755.803,E2 -15755.803} C_VEL
LIN {X 0,Y 312.746,Z 159.527,A -85,B 0,C 180,E1 -15759.051,E2 -15759.051} C_VEL
LIN {X 0,Y 312.601,Z 159.544,A -85,B 0,C 180,E1 -15762.993,E2 -15762.993} C_VEL
LIN {X 0,Y 312.542,Z 159.556,A -85,B 0,C 180,E1 -15765.655,E2 -15765.655} C_VEL
LIN {X 0,Y 312.514,Z 159.558,A -85,B 0,C 180,E1 -15769.715,E2 -15769.715} C_VEL
LIN {X 0,Y 312.509,Z 159.553,A -85,B 0,C 180,E1 -15772.775,E2 -15772.775} C_VEL
LIN {X 0,Y 312.478,Z 159.552,A -85,B 0,C 180,E1 -15776.733,E2 -15776.733} C_VEL
LIN {X 0,Y 312.465,Z 159.562,A -85,B 0,C 180,E1 -15779.659,E2 -15779.659} C_VEL
LIN {X 0,Y 312.517,Z 159.554,A -85,B 0,C 180,E1 -15783.69,E2 -15783.69} C_VEL
LIN {X 0,Y 312.51,Z 159.556,A -85,B 0,C 180,E1 -15787.388,E2 -15787.388} C_VEL
LIN {X 0,Y 312.438,Z 159.566,A -85,B 0,C 180,E1 -15790.718,E2 -15790.718} C_VEL
LIN {X 0,Y 312.424,Z 159.563,A -85,B 0,C 180,E1 -15791.497,E2 -15791.497} C_VEL
LIN {X 0,Y 311.773,Z 159.65,A -85,B 0,C 180,E1 -15792.573,E2 -15792.573} C_VEL
LIN {X 0,Y 308.914,Z 160.001,A -85,B 0,C 180,E1 -15794.324,E2 -15794.324} C_VEL
LIN {X 0,Y 306.498,Z 160.298,A -85,B 0,C 180,E1 -15795.745,E2 -15795.745} C_VEL
LIN {X 0,Y 305.489,Z 160.427,A -85,B 0,C 180,E1 -15796.845,E2 -15796.845} C_VEL
LIN {X 0,Y 305.422,Z 160.432,A -85,B 0,C 180,E1 -15797.218,E2 -15797.218} C_VEL
LIN {X 0,Y 305.459,Z 160.433,A -85,B 0,C 180,E1 -15801.596,E2 -15801.596} C_VEL
LIN {X 0,Y 305.461,Z 160.435,A -85,B 0,C 180,E1 -15804.888,E2 -15804.888} C_VEL
LIN {X 0,Y 305.442,Z 160.434,A -85,B 0,C 180,E1 -15808.359,E2 -15808.359} C_VEL
